// TIA Portal V17 export
// export: Created 2025-03-07T09:19:40.4759984Z, ExportSetting WithDefaults, DisplayName Totally Integrated Automation Portal, DisplayVersion V17 Update 8, DisplayName TIA Portal Openness, DisplayVersion V17 Update 8, DisplayName TIA Portal Version Control Interface, DisplayVersion V17, DisplayName SINAMICS Startdrive Advanced, DisplayVersion V17 SP2, DisplayName SINAMICS Startdrive G110M, G120, G120C, G120D, G120P, G115D, DisplayVersion V17 SP2, DisplayName SINAMICS Startdrive G130, G150, S120, S150, SINAMICS MV, S210, DisplayVersion V17 SP2, DisplayName STEP 7 Professional, DisplayVersion V17 Update 8, DisplayName SINUMERIK ONE STEP 7 Toolbox, DisplayVersion V17 Update 12, DisplayName SINUMERIK 840D sl STEP 7 Toolbox, DisplayVersion V17 Update 12, DisplayName STEP 7 Safety, DisplayVersion V17 Update 6, DisplayName WinCC Advanced, DisplayVersion V17 Update 8
TYPE "M_FUNCTIONS_FIXTURE"
// stored: IsFailsafeCompliant false
   STRUCT
      M_RESET_AUX : Bool;   // RESET AUX
      M_RESET_PULSE : Bool;   // RESET PULSE
      READ_IN_DISABLE_GENERAL : Bool;   // READ-IN DISABLE
      READ_IN_DISABLE_F1 : Bool;   // READ-IN DISABLE
      READ_IN_DISABLE_F2 : Bool;   // READ-IN DISABLE
      SPARE_05 : Bool;
      SPARE_06 : Bool;
      SPARE_07 : Bool;
      M0 : Bool;   // M0-PROGRAMMED STOP (SIEMENS)
      Ack_M0 : Bool;   // ACKNOWLEDGE M0-PROGRAMMED STOP (SIEMENS)
      M1 : Bool;   // M1-OPTIONAL STOP (SIEMENS)
      Ack_M1 : Bool;   // ACKNOWLEDGE M1-OPTIONAL STOP (SIEMENS)
      M2 : Bool;   // M2-END OF PROGRAM, MAIN PROGRAM, AS M30 (SIEMENS)
      Ack_M2 : Bool;   // ACKNOWLEDGE M2-END OF PROGRAM, MAIN PROGRAM, AS M30 (SIEMENS)
      M3 : Bool;   // M3-SPINDLE CLOCKWISE (SIEMENS)
      Ack_M3 : Bool;   // ACKNOWLEDGE M3-SPINDLE CLOCKWISE (SIEMENS)
      M4 : Bool;   // M4-SPINDLE COUNTER CLOCKWISE (SIEMENS)
      Ack_M4 : Bool;   // ACKNOWLEDGE M4-SPINDLE COUNTER CLOCKWISE (SIEMENS)
      M5 : Bool;   // M5-SPINDLE STOP (SIEMENS)
      Ack_M5 : Bool;   // ACKNOWLEDGE M5-SPINDLE STOP (SIEMENS)
      M6 : Bool;   // M6-TOOL CHANGE (SIEMENS)
      Ack_M6 : Bool;   // ACKNOWLEDGE M6-TOOL CHANGE (SIEMENS)
      M7 : Bool;   // M7-
      Ack_M7 : Bool;   // ACKNOWLEDGE M7-
      M8 : Bool;   // M8-
      Ack_M8 : Bool;   // ACKNOWLEDGE M8-
      M9 : Bool;   // M9-
      Ack_M9 : Bool;   // ACKNOWLEDGE M9-
      M10 : Bool;   // M10-
      Ack_M10 : Bool;   // ACKNOWLEDGE M10-
      M11 : Bool;   // M11-
      Ack_M11 : Bool;   // ACKNOWLEDGE M11-
      M12 : Bool;   // M12-
      Ack_M12 : Bool;   // ACKNOWLEDGE M12-
      M13 : Bool;   // M13-
      Ack_M13 : Bool;   // ACKNOWLEDGE M13-
      M14 : Bool;   // M14-
      Ack_M14 : Bool;   // ACKNOWLEDGE M14-
      M15 : Bool;   // M15-
      Ack_M15 : Bool;   // ACKNOWLEDGE M15-
      M16 : Bool;   // M16-
      Ack_M16 : Bool;   // ACKNOWLEDGE M16-
      M17 : Bool;   // M17-END OF SUBPROGRAM (SIEMENS)
      Ack_M17 : Bool;   // ACKNOWLEDGE M17-END OF SUBPROGRAM (SIEMENS)
      M18 : Bool;   // M18-
      Ack_M18 : Bool;   // ACKNOWLEDGE M18-
      M19 : Bool;   // M19-SPINDLE POSITIONING (SIEMENS)
      Ack_M19 : Bool;   // ACKNOWLEDGE M19-SPINDLE POSITIONING (SIEMENS)
      M20 : Bool;   // M20-
      Ack_M20 : Bool;   // ACKNOWLEDGE M20-
      M21 : Bool;   // M21-
      Ack_M21 : Bool;   // ACKNOWLEDGE M21-
      M22 : Bool;   // M22-
      Ack_M22 : Bool;   // ACKNOWLEDGE M22-
      M23 : Bool;   // M23-
      Ack_M23 : Bool;   // ACKNOWLEDGE M23-
      M24 : Bool;   // M24-
      Ack_M24 : Bool;   // ACKNOWLEDGE M24-
      M25 : Bool;   // M25-
      Ack_M25 : Bool;   // ACKNOWLEDGE M25-
      M26 : Bool;   // M26-
      Ack_M26 : Bool;   // ACKNOWLEDGE M26-
      M27 : Bool;   // M27-
      Ack_M27 : Bool;   // ACKNOWLEDGE M27-
      M28 : Bool;   // M28-
      Ack_M28 : Bool;   // ACKNOWLEDGE M28-
      M29 : Bool;   // M29-
      Ack_M29 : Bool;   // ACKNOWLEDGE M29-
      M30 : Bool;   // M30-END OF MAIN PROGRAM (SIEMENS)
      Ack_M30 : Bool;   // ACKNOWLEDGE M30-END OF MAIN PROGRAM (SIEMENS)
      M31 : Bool;   // M31-
      Ack_M31 : Bool;   // ACKNOWLEDGE M31-
      M32 : Bool;   // M32-
      Ack_M32 : Bool;   // ACKNOWLEDGE M32-
      M33 : Bool;   // M33-
      Ack_M33 : Bool;   // ACKNOWLEDGE M33-
      M34 : Bool;   // M34-
      Ack_M34 : Bool;   // ACKNOWLEDGE M34-
      M35 : Bool;   // M35-
      Ack_M35 : Bool;   // ACKNOWLEDGE M35-
      M36 : Bool;   // M36-
      Ack_M36 : Bool;   // ACKNOWLEDGE M36-
      M37 : Bool;   // M37-
      Ack_M37 : Bool;   // ACKNOWLEDGE M37-
      M38 : Bool;   // M38-
      Ack_M38 : Bool;   // ACKNOWLEDGE M38-
      M39 : Bool;   // M39-
      Ack_M39 : Bool;   // ACKNOWLEDGE M39-
      M40 : Bool;   // M40-AUTOMATIC GEAR CHANGE (SIEMENS)
      Ack_M40 : Bool;   // ACKNOWLEDGE M40-AUTOMATIC GEAR CHANGE (SIEMENS)
      M41 : Bool;   // M41-GEAR STAGE 1 (SIEMENS)
      Ack_M41 : Bool;   // ACKNOWLEDGE M41-GEAR STAGE 1 (SIEMENS)
      M42 : Bool;   // M42-GEAR STAGE 2 (SIEMENS)
      Ack_M42 : Bool;   // ACKNOWLEDGE M42-GEAR STAGE 2 (SIEMENS)
      M43 : Bool;   // M43-GEAR STAGE 3 (SIEMENS)
      Ack_M43 : Bool;   // ACKNOWLEDGE M43-GEAR STAGE 3 (SIEMENS)
      M44 : Bool;   // M44-GEAR STAGE 4 (SIEMENS)
      Ack_M44 : Bool;   // ACKNOWLEDGE M44-GEAR STAGE 4 (SIEMENS)
      M45 : Bool;   // M45-GEAR STAGE 5 (SIEMENS)
      Ack_M45 : Bool;   // ACKNOWLEDGE M45-GEAR STAGE 5 (SIEMENS)
      M46 : Bool;   // M46-
      Ack_M46 : Bool;   // ACKNOWLEDGE M46-
      M47 : Bool;   // M47-
      Ack_M47 : Bool;   // ACKNOWLEDGE M47-
      M48 : Bool;   // M48-
      Ack_M48 : Bool;   // ACKNOWLEDGE M48-
      M49 : Bool;   // M49-
      Ack_M49 : Bool;   // ACKNOWLEDGE M49-
      M50 : Bool;   // M50-
      Ack_M50 : Bool;   // ACKNOWLEDGE M50-
      M51 : Bool;   // M51-
      Ack_M51 : Bool;   // ACKNOWLEDGE M51-
      M52 : Bool;   // M52-
      Ack_M52 : Bool;   // ACKNOWLEDGE M52-
      M53 : Bool;   // M53-
      Ack_M53 : Bool;   // ACKNOWLEDGE M53-
      M54 : Bool;   // M54-
      Ack_M54 : Bool;   // ACKNOWLEDGE M54-
      M55 : Bool;   // M55-
      Ack_M55 : Bool;   // ACKNOWLEDGE M55-
      M56 : Bool;   // M56-
      Ack_M56 : Bool;   // ACKNOWLEDGE M56-
      M57 : Bool;   // M57-
      Ack_M57 : Bool;   // ACKNOWLEDGE M57-
      M58 : Bool;   // M58-
      Ack_M58 : Bool;   // ACKNOWLEDGE M58-
      M59 : Bool;   // M59-
      Ack_M59 : Bool;   // ACKNOWLEDGE M59-
      M60 : Bool;   // M60-
      Ack_M60 : Bool;   // ACKNOWLEDGE M60-
      M61 : Bool;   // M61-
      Ack_M61 : Bool;   // ACKNOWLEDGE M61-
      M62 : Bool;   // M62-
      Ack_M62 : Bool;   // ACKNOWLEDGE M62-
      M63 : Bool;   // M63-
      Ack_M63 : Bool;   // ACKNOWLEDGE M63-
      M64 : Bool;   // M64-
      Ack_M64 : Bool;   // ACKNOWLEDGE M64-
      M65 : Bool;   // M65-
      Ack_M65 : Bool;   // ACKNOWLEDGE M65-
      M66 : Bool;   // M66-
      Ack_M66 : Bool;   // ACKNOWLEDGE M66-
      M67 : Bool;   // M67-
      Ack_M67 : Bool;   // ACKNOWLEDGE M67-
      M68 : Bool;   // M68-
      Ack_M68 : Bool;   // ACKNOWLEDGE M68-
      M69 : Bool;   // M69-
      Ack_M69 : Bool;   // ACKNOWLEDGE M69-
      M70 : Bool;   // M70-SPINDLE IS SWITCHED TO AXIS MODE (SIEMENS)
      Ack_M70 : Bool;   // ACKNOWLEDGE M70-SPINDLE IS SWITCHED TO AXIS MODE (SIEMENS)
      M71 : Bool;   // M71-
      Ack_M71 : Bool;   // ACKNOWLEDGE M71-
      M72 : Bool;   // M72-
      Ack_M72 : Bool;   // ACKNOWLEDGE M72-
      M73 : Bool;   // M73-
      Ack_M73 : Bool;   // ACKNOWLEDGE M73-
      M74 : Bool;   // M74-
      Ack_M74 : Bool;   // ACKNOWLEDGE M74-
      M75 : Bool;   // M75-
      Ack_M75 : Bool;   // ACKNOWLEDGE M75-
      M76 : Bool;   // M76-
      Ack_M76 : Bool;   // ACKNOWLEDGE M76-
      M77 : Bool;   // M77-
      Ack_M77 : Bool;   // ACKNOWLEDGE M77-
      M78 : Bool;   // M78-
      Ack_M78 : Bool;   // ACKNOWLEDGE M78-
      M79 : Bool;   // M79-
      Ack_M79 : Bool;   // ACKNOWLEDGE M79-
      M80 : Bool;   // M80-
      Ack_M80 : Bool;   // ACKNOWLEDGE M80-
      M81 : Bool;   // M81-
      Ack_M81 : Bool;   // ACKNOWLEDGE M81-
      M82 : Bool;   // M82-
      Ack_M82 : Bool;   // ACKNOWLEDGE M82-
      M83 : Bool;   // M83-
      Ack_M83 : Bool;   // ACKNOWLEDGE M83-
      M84 : Bool;   // M84-
      Ack_M84 : Bool;   // ACKNOWLEDGE M84-
      M85 : Bool;   // M85-
      Ack_M85 : Bool;   // ACKNOWLEDGE M85-
      M86 : Bool;   // M86-
      Ack_M86 : Bool;   // ACKNOWLEDGE M86-
      M87 : Bool;   // M87-
      Ack_M87 : Bool;   // ACKNOWLEDGE M87-
      M88 : Bool;   // M88-
      Ack_M88 : Bool;   // ACKNOWLEDGE M88-
      M89 : Bool;   // M89-
      Ack_M89 : Bool;   // ACKNOWLEDGE M89-
      M90 : Bool;   // M90-
      Ack_M90 : Bool;   // ACKNOWLEDGE M90-
      M91 : Bool;   // M91-
      Ack_M91 : Bool;   // ACKNOWLEDGE M91-
      M92 : Bool;   // M92-
      Ack_M92 : Bool;   // ACKNOWLEDGE M92-
      M93 : Bool;   // M93-
      Ack_M93 : Bool;   // ACKNOWLEDGE M93-
      M94 : Bool;   // M94-
      Ack_M94 : Bool;   // ACKNOWLEDGE M94-
      M95 : Bool;   // M95-
      Ack_M95 : Bool;   // ACKNOWLEDGE M95-
      M96 : Bool;   // M96-
      Ack_M96 : Bool;   // ACKNOWLEDGE M96-
      M97 : Bool;   // M97-
      Ack_M97 : Bool;   // ACKNOWLEDGE M97-
      M98 : Bool;   // M98-EXTERNAL LANGUAGE (SIEMENS)
      Ack_M98 : Bool;   // ACKNOWLEDGE M98-EXTERNAL LANGUAGE (SIEMENS)
      M99 : Bool;   // M99-EXTERNAL LANGUAGE (SIEMENS)
      Ack_M99 : Bool;   // ACKNOWLEDGE M99-EXTERNAL LANGUAGE (SIEMENS)
      M100 : Bool;   // M100-FIXTURE WAITS FULL DEPTHS UNIT 01R (READ-IN DISABLE)
      Ack_M100 : Bool;   // ACKNOWLEDGE M100-FIXTURE WAITS FULL DEPTHS UNIT 01R (READ-IN DISABLE)
      M101 : Bool;   // M101-FIXTURE WAITS FULL DEPTHS UNIT 01L (READ-IN DISABLE)
      Ack_M101 : Bool;   // ACKNOWLEDGE M101-FIXTURE WAITS FULL DEPTHS UNIT 01L (READ-IN DISABLE)
      M102 : Bool;   // M102-AXIS B IN POSITION DURING LOAD-UNLOAD (READ-IN DISABLE)
      Ack_M102 : Bool;   // ACKNOWLEDGE M102-AXIS B IN POSITION DURING LOAD-UNLOAD (READ-IN DISABLE)
      M103 : Bool;   // M103-
      Ack_M103 : Bool;   // ACKNOWLEDGE M103-
      M104 : Bool;   // M104-
      Ack_M104 : Bool;   // ACKNOWLEDGE M104-
      M105 : Bool;   // M105-
      Ack_M105 : Bool;   // ACKNOWLEDGE M105-
      M106 : Bool;   // M106-
      Ack_M106 : Bool;   // ACKNOWLEDGE M106-
      M107 : Bool;   // M107-
      Ack_M107 : Bool;   // ACKNOWLEDGE M107-
      M108 : Bool;   // M108-
      Ack_M108 : Bool;   // ACKNOWLEDGE M108-
      M109 : Bool;   // M109-
      Ack_M109 : Bool;   // ACKNOWLEDGE M109-
      M110 : Bool;   // M110-UNBLOCK TABLE
      Ack_M110 : Bool;   // ACKNOWLEDGE M110-UNBLOCK TABLE
      M111 : Bool;   // M111-BLOCK TABLE
      Ack_M111 : Bool;   // ACKNOWLEDGE M111-BLOCK TABLE
      M112 : Bool;   // M112-
      Ack_M112 : Bool;   // ACKNOWLEDGE M112-
      M113 : Bool;   // M113-
      Ack_M113 : Bool;   // ACKNOWLEDGE M113-
      M114 : Bool;   // M114-
      Ack_M114 : Bool;   // ACKNOWLEDGE M114-
      M115 : Bool;   // M115-
      Ack_M115 : Bool;   // ACKNOWLEDGE M115-
      M116 : Bool;   // M116-
      Ack_M116 : Bool;   // ACKNOWLEDGE M116-
      M117 : Bool;   // M117-
      Ack_M117 : Bool;   // ACKNOWLEDGE M117-
      M118 : Bool;   // M118-
      Ack_M118 : Bool;   // ACKNOWLEDGE M118-
      M119 : Bool;   // M119-
      Ack_M119 : Bool;   // ACKNOWLEDGE M119-
      M120 : Bool;   // M120-
      Ack_M120 : Bool;   // ACKNOWLEDGE M120-
      M121 : Bool;   // M121-
      Ack_M121 : Bool;   // ACKNOWLEDGE M121-
      M122 : Bool;   // M122-
      Ack_M122 : Bool;   // ACKNOWLEDGE M122-
      M123 : Bool;   // M123-AXIS B TORQUE LIMIT EXCEEDED
      Ack_M123 : Bool;   // ACKNOWLEDGE M123-AXIS B TORQUE LIMIT EXCEEDED
      M124 : Bool;   // M124-
      Ack_M124 : Bool;   // ACKNOWLEDGE M124-
      M125 : Bool;   // M125-
      Ack_M125 : Bool;   // ACKNOWLEDGE M125-
      M126 : Bool;   // M126-
      Ack_M126 : Bool;   // ACKNOWLEDGE M126-
      M127 : Bool;   // M127-
      Ack_M127 : Bool;   // ACKNOWLEDGE M127-
      M128 : Bool;   // M128-
      Ack_M128 : Bool;   // ACKNOWLEDGE M128-
      M129 : Bool;   // M129-
      Ack_M129 : Bool;   // ACKNOWLEDGE M129-
      M130 : Bool;   // M130-
      Ack_M130 : Bool;   // ACKNOWLEDGE M130-
      M131 : Bool;   // M131-
      Ack_M131 : Bool;   // ACKNOWLEDGE M131-
      M132 : Bool;   // M132-
      Ack_M132 : Bool;   // ACKNOWLEDGE M132-
      M133 : Bool;   // M133-
      Ack_M133 : Bool;   // ACKNOWLEDGE M133-
      M134 : Bool;   // M134-
      Ack_M134 : Bool;   // ACKNOWLEDGE M134-
      M135 : Bool;   // M135-
      Ack_M135 : Bool;   // ACKNOWLEDGE M135-
      M136 : Bool;   // M136-
      Ack_M136 : Bool;   // ACKNOWLEDGE M136-
      M137 : Bool;   // M137-
      Ack_M137 : Bool;   // ACKNOWLEDGE M137-
      M138 : Bool;   // M138-
      Ack_M138 : Bool;   // ACKNOWLEDGE M138-
      M139 : Bool;   // M139-
      Ack_M139 : Bool;   // ACKNOWLEDGE M139-
      M140 : Bool;   // M140-
      Ack_M140 : Bool;   // ACKNOWLEDGE M140-
      M141 : Bool;   // M141-
      Ack_M141 : Bool;   // ACKNOWLEDGE M141-
      M142 : Bool;   // M142-
      Ack_M142 : Bool;   // ACKNOWLEDGE M142-
      M143 : Bool;   // M143-
      Ack_M143 : Bool;   // ACKNOWLEDGE M143-
      M144 : Bool;   // M144-
      Ack_M144 : Bool;   // ACKNOWLEDGE M144-
      M145 : Bool;   // M145-
      Ack_M145 : Bool;   // ACKNOWLEDGE M145-
      M146 : Bool;   // M146-
      Ack_M146 : Bool;   // ACKNOWLEDGE M146-
      M147 : Bool;   // M147-
      Ack_M147 : Bool;   // ACKNOWLEDGE M147-
      M148 : Bool;   // M148-
      Ack_M148 : Bool;   // ACKNOWLEDGE M148-
      M149 : Bool;   // M149-
      Ack_M149 : Bool;   // ACKNOWLEDGE M149-
      M150 : Bool;   // M150-AUTOMATIC DOOR OPEN
      Ack_M150 : Bool;   // ACKNOWLEDGE M150-AUTOMATIC DOOR OPEN
      M151 : Bool;   // M151-AUTOMATIC DOOR CLOSE
      Ack_M151 : Bool;   // ACKNOWLEDGE M151-AUTOMATIC DOOR CLOSE
      M152 : Bool;   // M152-
      Ack_M152 : Bool;   // ACKNOWLEDGE M152-
      M153 : Bool;   // M153-
      Ack_M153 : Bool;   // ACKNOWLEDGE M153-
      M154 : Bool;   // M154-
      Ack_M154 : Bool;   // ACKNOWLEDGE M154-
      M155 : Bool;   // M155-
      Ack_M155 : Bool;   // ACKNOWLEDGE M155-
      M156 : Bool;   // M156-
      Ack_M156 : Bool;   // ACKNOWLEDGE M156-
      M157 : Bool;   // M157-
      Ack_M157 : Bool;   // ACKNOWLEDGE M157-
      M158 : Bool;   // M158-
      Ack_M158 : Bool;   // ACKNOWLEDGE M158-
      M159 : Bool;   // M159-
      Ack_M159 : Bool;   // ACKNOWLEDGE M159-
      M160 : Bool;   // M160-
      Ack_M160 : Bool;   // ACKNOWLEDGE M160-
      M161 : Bool;   // M161-
      Ack_M161 : Bool;   // ACKNOWLEDGE M161-
      M162 : Bool;   // M162-
      Ack_M162 : Bool;   // ACKNOWLEDGE M162-
      M163 : Bool;   // M163-
      Ack_M163 : Bool;   // ACKNOWLEDGE M163-
      M164 : Bool;   // M164-
      Ack_M164 : Bool;   // ACKNOWLEDGE M164-
      M165 : Bool;   // M165-
      Ack_M165 : Bool;   // ACKNOWLEDGE M165-
      M166 : Bool;   // M166-
      Ack_M166 : Bool;   // ACKNOWLEDGE M166-
      M167 : Bool;   // M167-
      Ack_M167 : Bool;   // ACKNOWLEDGE M167-
      M168 : Bool;   // M168-
      Ack_M168 : Bool;   // ACKNOWLEDGE M168-
      M169 : Bool;   // M169-
      Ack_M169 : Bool;   // ACKNOWLEDGE M169-
      M170 : Bool;   // M170-
      Ack_M170 : Bool;   // ACKNOWLEDGE M170-
      M171 : Bool;   // M171-
      Ack_M171 : Bool;   // ACKNOWLEDGE M171-
      M172 : Bool;   // M172-
      Ack_M172 : Bool;   // ACKNOWLEDGE M172-
      M173 : Bool;   // M173-
      Ack_M173 : Bool;   // ACKNOWLEDGE M173-
      M174 : Bool;   // M174-
      Ack_M174 : Bool;   // ACKNOWLEDGE M174-
      M175 : Bool;   // M175-
      Ack_M175 : Bool;   // ACKNOWLEDGE M175-
      M176 : Bool;   // M176-
      Ack_M176 : Bool;   // ACKNOWLEDGE M176-
      M177 : Bool;   // M177-
      Ack_M177 : Bool;   // ACKNOWLEDGE M177-
      M178 : Bool;   // M178-
      Ack_M178 : Bool;   // ACKNOWLEDGE M178-
      M179 : Bool;   // M179-
      Ack_M179 : Bool;   // ACKNOWLEDGE M179-
      M180 : Bool;   // M180-
      Ack_M180 : Bool;   // ACKNOWLEDGE M180-
      M181 : Bool;   // M181-
      Ack_M181 : Bool;   // ACKNOWLEDGE M181-
      M182 : Bool;   // M182-
      Ack_M182 : Bool;   // ACKNOWLEDGE M182-
      M183 : Bool;   // M183-
      Ack_M183 : Bool;   // ACKNOWLEDGE M183-
      M184 : Bool;   // M184-
      Ack_M184 : Bool;   // ACKNOWLEDGE M184-
      M185 : Bool;   // M185-
      Ack_M185 : Bool;   // ACKNOWLEDGE M185-
      M186 : Bool;   // M186-
      Ack_M186 : Bool;   // ACKNOWLEDGE M186-
      M187 : Bool;   // M187-
      Ack_M187 : Bool;   // ACKNOWLEDGE M187-
      M188 : Bool;   // M188-
      Ack_M188 : Bool;   // ACKNOWLEDGE M188-
      M189 : Bool;   // M189-
      Ack_M189 : Bool;   // ACKNOWLEDGE M189-
      M190 : Bool;   // M190-
      Ack_M190 : Bool;   // ACKNOWLEDGE M190-
      M191 : Bool;   // M191-
      Ack_M191 : Bool;   // ACKNOWLEDGE M191-
      M192 : Bool;   // M192-
      Ack_M192 : Bool;   // ACKNOWLEDGE M192-
      M193 : Bool;   // M193-
      Ack_M193 : Bool;   // ACKNOWLEDGE M193-
      M194 : Bool;   // M194-
      Ack_M194 : Bool;   // ACKNOWLEDGE M194-
      M195 : Bool;   // M195-
      Ack_M195 : Bool;   // ACKNOWLEDGE M195-
      M196 : Bool;   // M196-
      Ack_M196 : Bool;   // ACKNOWLEDGE M196-
      M197 : Bool;   // M197-
      Ack_M197 : Bool;   // ACKNOWLEDGE M197-
      M198 : Bool;   // M198-
      Ack_M198 : Bool;   // ACKNOWLEDGE M198-
      M199 : Bool;   // M199-
      Ack_M199 : Bool;   // ACKNOWLEDGE M199-
      M200 : Bool;   // M200-
      Ack_M200 : Bool;   // ACKNOWLEDGE M200-
      M201 : Bool;   // M201-
      Ack_M201 : Bool;   // ACKNOWLEDGE M201-
      M202 : Bool;   // M202-
      Ack_M202 : Bool;   // ACKNOWLEDGE M202-
      M203 : Bool;   // M203-
      Ack_M203 : Bool;   // ACKNOWLEDGE M203-
      M204 : Bool;   // M204-
      Ack_M204 : Bool;   // ACKNOWLEDGE M204-
      M205 : Bool;   // M205-
      Ack_M205 : Bool;   // ACKNOWLEDGE M205-
      M206 : Bool;   // M206-
      Ack_M206 : Bool;   // ACKNOWLEDGE M206-
      M207 : Bool;   // M207-
      Ack_M207 : Bool;   // ACKNOWLEDGE M207-
      M208 : Bool;   // M208-
      Ack_M208 : Bool;   // ACKNOWLEDGE M208-
      M209 : Bool;   // M209-
      Ack_M209 : Bool;   // ACKNOWLEDGE M209-
      M210 : Bool;   // M210-
      Ack_M210 : Bool;   // ACKNOWLEDGE M210-
      M211 : Bool;   // M211-
      Ack_M211 : Bool;   // ACKNOWLEDGE M211-
      M212 : Bool;   // M212-
      Ack_M212 : Bool;   // ACKNOWLEDGE M212-
      M213 : Bool;   // M213-
      Ack_M213 : Bool;   // ACKNOWLEDGE M213-
      M214 : Bool;   // M214-
      Ack_M214 : Bool;   // ACKNOWLEDGE M214-
      M215 : Bool;   // M215-
      Ack_M215 : Bool;   // ACKNOWLEDGE M215-
      M216 : Bool;   // M216-
      Ack_M216 : Bool;   // ACKNOWLEDGE M216-
      M217 : Bool;   // M217-
      Ack_M217 : Bool;   // ACKNOWLEDGE M217-
      M218 : Bool;   // M218-
      Ack_M218 : Bool;   // ACKNOWLEDGE M218-
      M219 : Bool;   // M219-
      Ack_M219 : Bool;   // ACKNOWLEDGE M219-
      M220 : Bool;   // M220-
      Ack_M220 : Bool;   // ACKNOWLEDGE M220-
      M221 : Bool;   // M221-
      Ack_M221 : Bool;   // ACKNOWLEDGE M221-
      M222 : Bool;   // M222-
      Ack_M222 : Bool;   // ACKNOWLEDGE M222-
      M223 : Bool;   // M223-
      Ack_M223 : Bool;   // ACKNOWLEDGE M223-
      M224 : Bool;   // M224-
      Ack_M224 : Bool;   // ACKNOWLEDGE M224-
      M225 : Bool;   // M225-
      Ack_M225 : Bool;   // ACKNOWLEDGE M225-
      M226 : Bool;   // M226-
      Ack_M226 : Bool;   // ACKNOWLEDGE M226-
      M227 : Bool;   // M227-
      Ack_M227 : Bool;   // ACKNOWLEDGE M227-
      M228 : Bool;   // M228-
      Ack_M228 : Bool;   // ACKNOWLEDGE M228-
      M229 : Bool;   // M229-
      Ack_M229 : Bool;   // ACKNOWLEDGE M229-
      M230 : Bool;   // M230-
      Ack_M230 : Bool;   // ACKNOWLEDGE M230-
      M231 : Bool;   // M231-
      Ack_M231 : Bool;   // ACKNOWLEDGE M231-
      M232 : Bool;   // M232-
      Ack_M232 : Bool;   // ACKNOWLEDGE M232-
      M233 : Bool;   // M233-
      Ack_M233 : Bool;   // ACKNOWLEDGE M233-
      M234 : Bool;   // M234-
      Ack_M234 : Bool;   // ACKNOWLEDGE M234-
      M235 : Bool;   // M235-
      Ack_M235 : Bool;   // ACKNOWLEDGE M235-
      M236 : Bool;   // M236-
      Ack_M236 : Bool;   // ACKNOWLEDGE M236-
      M237 : Bool;   // M237-
      Ack_M237 : Bool;   // ACKNOWLEDGE M237-
      M238 : Bool;   // M238-
      Ack_M238 : Bool;   // ACKNOWLEDGE M238-
      M239 : Bool;   // M239-
      Ack_M239 : Bool;   // ACKNOWLEDGE M239-
      M240 : Bool;   // M240-
      Ack_M240 : Bool;   // ACKNOWLEDGE M240-
      M241 : Bool;   // M241-
      Ack_M241 : Bool;   // ACKNOWLEDGE M241-
      M242 : Bool;   // M242-
      Ack_M242 : Bool;   // ACKNOWLEDGE M242-
      M243 : Bool;   // M243-
      Ack_M243 : Bool;   // ACKNOWLEDGE M243-
      M244 : Bool;   // M244-
      Ack_M244 : Bool;   // ACKNOWLEDGE M244-
      M245 : Bool;   // M245-
      Ack_M245 : Bool;   // ACKNOWLEDGE M245-
      M246 : Bool;   // M246-
      Ack_M246 : Bool;   // ACKNOWLEDGE M246-
      M247 : Bool;   // M247-
      Ack_M247 : Bool;   // ACKNOWLEDGE M247-
      M248 : Bool;   // M248-
      Ack_M248 : Bool;   // ACKNOWLEDGE M248-
      M249 : Bool;   // M249-
      Ack_M249 : Bool;   // ACKNOWLEDGE M249-
      M250 : Bool;   // M250-
      Ack_M250 : Bool;   // ACKNOWLEDGE M250-
      M251 : Bool;   // M251-
      Ack_M251 : Bool;   // ACKNOWLEDGE M251-
      M252 : Bool;   // M252-
      Ack_M252 : Bool;   // ACKNOWLEDGE M252-
      M253 : Bool;   // M253-
      Ack_M253 : Bool;   // ACKNOWLEDGE M253-
      M254 : Bool;   // M254-
      Ack_M254 : Bool;   // ACKNOWLEDGE M254-
      M255 : Bool;   // M255-
      Ack_M255 : Bool;   // ACKNOWLEDGE M255-
      M256 : Bool;   // M256-
      Ack_M256 : Bool;   // ACKNOWLEDGE M256-
      M257 : Bool;   // M257-
      Ack_M257 : Bool;   // ACKNOWLEDGE M257-
      M258 : Bool;   // M258-
      Ack_M258 : Bool;   // ACKNOWLEDGE M258-
      M259 : Bool;   // M259-
      Ack_M259 : Bool;   // ACKNOWLEDGE M259-
      M260 : Bool;   // M260-
      Ack_M260 : Bool;   // ACKNOWLEDGE M260-
      M261 : Bool;   // M261-
      Ack_M261 : Bool;   // ACKNOWLEDGE M261-
      M262 : Bool;   // M262-
      Ack_M262 : Bool;   // ACKNOWLEDGE M262-
      M263 : Bool;   // M263-
      Ack_M263 : Bool;   // ACKNOWLEDGE M263-
      M264 : Bool;   // M264-
      Ack_M264 : Bool;   // ACKNOWLEDGE M264-
      M265 : Bool;   // M265-
      Ack_M265 : Bool;   // ACKNOWLEDGE M265-
      M266 : Bool;   // M266-
      Ack_M266 : Bool;   // ACKNOWLEDGE M266-
      M267 : Bool;   // M267-
      Ack_M267 : Bool;   // ACKNOWLEDGE M267-
      M268 : Bool;   // M268-
      Ack_M268 : Bool;   // ACKNOWLEDGE M268-
      M269 : Bool;   // M269-
      Ack_M269 : Bool;   // ACKNOWLEDGE M269-
      M270 : Bool;   // M270-
      Ack_M270 : Bool;   // ACKNOWLEDGE M270-
      M271 : Bool;   // M271-
      Ack_M271 : Bool;   // ACKNOWLEDGE M271-
      M272 : Bool;   // M272-
      Ack_M272 : Bool;   // ACKNOWLEDGE M272-
      M273 : Bool;   // M273-
      Ack_M273 : Bool;   // ACKNOWLEDGE M273-
      M274 : Bool;   // M274-
      Ack_M274 : Bool;   // ACKNOWLEDGE M274-
      M275 : Bool;   // M275-
      Ack_M275 : Bool;   // ACKNOWLEDGE M275-
      M276 : Bool;   // M276-
      Ack_M276 : Bool;   // ACKNOWLEDGE M276-
      M277 : Bool;   // M277-
      Ack_M277 : Bool;   // ACKNOWLEDGE M277-
      M278 : Bool;   // M278-
      Ack_M278 : Bool;   // ACKNOWLEDGE M278-
      M279 : Bool;   // M279-
      Ack_M279 : Bool;   // ACKNOWLEDGE M279-
      M280 : Bool;   // M280-
      Ack_M280 : Bool;   // ACKNOWLEDGE M280-
      M281 : Bool;   // M281-
      Ack_M281 : Bool;   // ACKNOWLEDGE M281-
      M282 : Bool;   // M282-
      Ack_M282 : Bool;   // ACKNOWLEDGE M282-
      M283 : Bool;   // M283-
      Ack_M283 : Bool;   // ACKNOWLEDGE M283-
      M284 : Bool;   // M284-
      Ack_M284 : Bool;   // ACKNOWLEDGE M284-
      M285 : Bool;   // M285-
      Ack_M285 : Bool;   // ACKNOWLEDGE M285-
      M286 : Bool;   // M286-
      Ack_M286 : Bool;   // ACKNOWLEDGE M286-
      M287 : Bool;   // M287-
      Ack_M287 : Bool;   // ACKNOWLEDGE M287-
      M288 : Bool;   // M288-
      Ack_M288 : Bool;   // ACKNOWLEDGE M288-
      M289 : Bool;   // M289-
      Ack_M289 : Bool;   // ACKNOWLEDGE M289-
      M290 : Bool;   // M290-
      Ack_M290 : Bool;   // ACKNOWLEDGE M290-
      M291 : Bool;   // M291-
      Ack_M291 : Bool;   // ACKNOWLEDGE M291-
      M292 : Bool;   // M292-
      Ack_M292 : Bool;   // ACKNOWLEDGE M292-
      M293 : Bool;   // M293-
      Ack_M293 : Bool;   // ACKNOWLEDGE M293-
      M294 : Bool;   // M294-
      Ack_M294 : Bool;   // ACKNOWLEDGE M294-
      M295 : Bool;   // M295-
      Ack_M295 : Bool;   // ACKNOWLEDGE M295-
      M296 : Bool;   // M296-
      Ack_M296 : Bool;   // ACKNOWLEDGE M296-
      M297 : Bool;   // M297-
      Ack_M297 : Bool;   // ACKNOWLEDGE M297-
      M298 : Bool;   // M298-
      Ack_M298 : Bool;   // ACKNOWLEDGE M298-
      M299 : Bool;   // M299-
      Ack_M299 : Bool;   // ACKNOWLEDGE M299-
      M300 : Bool;   // M300-
      Ack_M300 : Bool;   // ACKNOWLEDGE M300-
      M301 : Bool;   // M301-
      Ack_M301 : Bool;   // ACKNOWLEDGE M301-
      M302 : Bool;   // M302-
      Ack_M302 : Bool;   // ACKNOWLEDGE M302-
      M303 : Bool;   // M303-
      Ack_M303 : Bool;   // ACKNOWLEDGE M303-
      M304 : Bool;   // M304-
      Ack_M304 : Bool;   // ACKNOWLEDGE M304-
      M305 : Bool;   // M305-
      Ack_M305 : Bool;   // ACKNOWLEDGE M305-
      M306 : Bool;   // M306-
      Ack_M306 : Bool;   // ACKNOWLEDGE M306-
      M307 : Bool;   // M307-
      Ack_M307 : Bool;   // ACKNOWLEDGE M307-
      M308 : Bool;   // M308-
      Ack_M308 : Bool;   // ACKNOWLEDGE M308-
      M309 : Bool;   // M309-
      Ack_M309 : Bool;   // ACKNOWLEDGE M309-
      M310 : Bool;   // M310-
      Ack_M310 : Bool;   // ACKNOWLEDGE M310-
      M311 : Bool;   // M311-
      Ack_M311 : Bool;   // ACKNOWLEDGE M311-
      M312 : Bool;   // M312-
      Ack_M312 : Bool;   // ACKNOWLEDGE M312-
      M313 : Bool;   // M313-
      Ack_M313 : Bool;   // ACKNOWLEDGE M313-
      M314 : Bool;   // M314-
      Ack_M314 : Bool;   // ACKNOWLEDGE M314-
      M315 : Bool;   // M315-
      Ack_M315 : Bool;   // ACKNOWLEDGE M315-
      M316 : Bool;   // M316-
      Ack_M316 : Bool;   // ACKNOWLEDGE M316-
      M317 : Bool;   // M317-
      Ack_M317 : Bool;   // ACKNOWLEDGE M317-
      M318 : Bool;   // M318-
      Ack_M318 : Bool;   // ACKNOWLEDGE M318-
      M319 : Bool;   // M319-
      Ack_M319 : Bool;   // ACKNOWLEDGE M319-
      M320 : Bool;   // M320-MACHINE FLUSH VALVE SWITCH ON
      Ack_M320 : Bool;   // ACKNOWLEDGE M320-MACHINE FLUSH VALVE SWITCH ON
      M321 : Bool;   // M321-MACHINE FLUSH VALVE SWITCH OFF
      Ack_M321 : Bool;   // ACKNOWLEDGE M321-MACHINE FLUSH VALVE SWITCH OFF
      M322 : Bool;   // M322-
      Ack_M322 : Bool;   // ACKNOWLEDGE M322-
      M323 : Bool;   // M323-
      Ack_M323 : Bool;   // ACKNOWLEDGE M323-
      M324 : Bool;   // M324-FIXTURE 1 CLEANING VALVE SWITCH ON
      Ack_M324 : Bool;   // ACKNOWLEDGE M324-FIXTURE 1 CLEANING VALVE SWITCH ON
      M325 : Bool;   // M325-FIXTURE 1 CLEANING VALVE SWITCH OFF
      Ack_M325 : Bool;   // ACKNOWLEDGE M325-FIXTURE 1 CLEANING VALVE SWITCH OFF
      M326 : Bool;   // M326-FIXTURE 2 CLEANING VALVE SWITCH ON
      Ack_M326 : Bool;   // ACKNOWLEDGE M326-FIXTURE 2 CLEANING VALVE SWITCH ON
      M327 : Bool;   // M327-FIXTURE 2 CLEANING VALVE SWITCH OFF
      Ack_M327 : Bool;   // ACKNOWLEDGE M327-FIXTURE 2 CLEANING VALVE SWITCH OFF
      M328 : Bool;   // M328-
      Ack_M328 : Bool;   // ACKNOWLEDGE M328-
      M329 : Bool;   // M329-
      Ack_M329 : Bool;   // ACKNOWLEDGE M329-
      M330 : Bool;   // M330-
      Ack_M330 : Bool;   // ACKNOWLEDGE M330-
      M331 : Bool;   // M331-
      Ack_M331 : Bool;   // ACKNOWLEDGE M331-
      M332 : Bool;   // M332-FIXTURE 1 INTERNAL BLOWING SWITCH ON
      Ack_M332 : Bool;   // ACKNOWLEDGE M332-FIXTURE 1 INTERNAL BLOWING SWITCH ON
      M333 : Bool;   // M333-FIXTURE 1 INTERNAL BLOWING SWITCH OFF
      Ack_M333 : Bool;   // ACKNOWLEDGE M333-FIXTURE 1 INTERNAL BLOWING SWITCH OFF
      M334 : Bool;   // M334-FIXTURE 2 INTERNAL BLOWING SWITCH ON
      Ack_M334 : Bool;   // ACKNOWLEDGE M334-FIXTURE 2 INTERNAL BLOWING SWITCH ON
      M335 : Bool;   // M335-FIXTURE 2 INTERNAL BLOWING SWITCH OFF
      Ack_M335 : Bool;   // ACKNOWLEDGE M335-FIXTURE 2 INTERNAL BLOWING SWITCH OFF
      M336 : Bool;   // M336-
      Ack_M336 : Bool;   // ACKNOWLEDGE M336-
      M337 : Bool;   // M337-
      Ack_M337 : Bool;   // ACKNOWLEDGE M337-
      M338 : Bool;   // M338-
      Ack_M338 : Bool;   // ACKNOWLEDGE M338-
      M339 : Bool;   // M339-
      Ack_M339 : Bool;   // ACKNOWLEDGE M339-
      M340 : Bool;   // M340-
      Ack_M340 : Bool;   // ACKNOWLEDGE M340-
      M341 : Bool;   // M341-
      Ack_M341 : Bool;   // ACKNOWLEDGE M341-
      M342 : Bool;   // M342-
      Ack_M342 : Bool;   // ACKNOWLEDGE M342-
      M343 : Bool;   // M343-
      Ack_M343 : Bool;   // ACKNOWLEDGE M343-
      M344 : Bool;   // M344-
      Ack_M344 : Bool;   // ACKNOWLEDGE M344-
      M345 : Bool;   // M345-
      Ack_M345 : Bool;   // ACKNOWLEDGE M345-
      M346 : Bool;   // M346-
      Ack_M346 : Bool;   // ACKNOWLEDGE M346-
      M347 : Bool;   // M347-
      Ack_M347 : Bool;   // ACKNOWLEDGE M347-
      M348 : Bool;   // M348-
      Ack_M348 : Bool;   // ACKNOWLEDGE M348-
      M349 : Bool;   // M349-
      Ack_M349 : Bool;   // ACKNOWLEDGE M349-
      M350 : Bool;   // M350-
      Ack_M350 : Bool;   // ACKNOWLEDGE M350-
      M351 : Bool;   // M351-
      Ack_M351 : Bool;   // ACKNOWLEDGE M351-
      M352 : Bool;   // M352-
      Ack_M352 : Bool;   // ACKNOWLEDGE M352-
      M353 : Bool;   // M353-
      Ack_M353 : Bool;   // ACKNOWLEDGE M353-
      M354 : Bool;   // M354-
      Ack_M354 : Bool;   // ACKNOWLEDGE M354-
      M355 : Bool;   // M355-
      Ack_M355 : Bool;   // ACKNOWLEDGE M355-
      M356 : Bool;   // M356-
      Ack_M356 : Bool;   // ACKNOWLEDGE M356-
      M357 : Bool;   // M357-
      Ack_M357 : Bool;   // ACKNOWLEDGE M357-
      M358 : Bool;   // M358-
      Ack_M358 : Bool;   // ACKNOWLEDGE M358-
      M359 : Bool;   // M359-
      Ack_M359 : Bool;   // ACKNOWLEDGE M359-
      M360 : Bool;   // M360-
      Ack_M360 : Bool;   // ACKNOWLEDGE M360-
      M361 : Bool;   // M361-
      Ack_M361 : Bool;   // ACKNOWLEDGE M361-
      M362 : Bool;   // M362-
      Ack_M362 : Bool;   // ACKNOWLEDGE M362-
      M363 : Bool;   // M363-
      Ack_M363 : Bool;   // ACKNOWLEDGE M363-
      M364 : Bool;   // M364-
      Ack_M364 : Bool;   // ACKNOWLEDGE M364-
      M365 : Bool;   // M365-
      Ack_M365 : Bool;   // ACKNOWLEDGE M365-
      M366 : Bool;   // M366-
      Ack_M366 : Bool;   // ACKNOWLEDGE M366-
      M367 : Bool;   // M367-
      Ack_M367 : Bool;   // ACKNOWLEDGE M367-
      M368 : Bool;   // M368-
      Ack_M368 : Bool;   // ACKNOWLEDGE M368-
      M369 : Bool;   // M369-
      Ack_M369 : Bool;   // ACKNOWLEDGE M369-
      M370 : Bool;   // M370-
      Ack_M370 : Bool;   // ACKNOWLEDGE M370-
      M371 : Bool;   // M371-
      Ack_M371 : Bool;   // ACKNOWLEDGE M371-
      M372 : Bool;   // M372-
      Ack_M372 : Bool;   // ACKNOWLEDGE M372-
      M373 : Bool;   // M373-
      Ack_M373 : Bool;   // ACKNOWLEDGE M373-
      M374 : Bool;   // M374-
      Ack_M374 : Bool;   // ACKNOWLEDGE M374-
      M375 : Bool;   // M375-
      Ack_M375 : Bool;   // ACKNOWLEDGE M375-
      M376 : Bool;   // M376-
      Ack_M376 : Bool;   // ACKNOWLEDGE M376-
      M377 : Bool;   // M377-
      Ack_M377 : Bool;   // ACKNOWLEDGE M377-
      M378 : Bool;   // M378-
      Ack_M378 : Bool;   // ACKNOWLEDGE M378-
      M379 : Bool;   // M379-
      Ack_M379 : Bool;   // ACKNOWLEDGE M379-
      M380 : Bool;   // M380-
      Ack_M380 : Bool;   // ACKNOWLEDGE M380-
      M381 : Bool;   // M381-
      Ack_M381 : Bool;   // ACKNOWLEDGE M381-
      M382 : Bool;   // M382-
      Ack_M382 : Bool;   // ACKNOWLEDGE M382-
      M383 : Bool;   // M383-
      Ack_M383 : Bool;   // ACKNOWLEDGE M383-
      M384 : Bool;   // M384-
      Ack_M384 : Bool;   // ACKNOWLEDGE M384-
      M385 : Bool;   // M385-
      Ack_M385 : Bool;   // ACKNOWLEDGE M385-
      M386 : Bool;   // M386-
      Ack_M386 : Bool;   // ACKNOWLEDGE M386-
      M387 : Bool;   // M387-
      Ack_M387 : Bool;   // ACKNOWLEDGE M387-
      M388 : Bool;   // M388-
      Ack_M388 : Bool;   // ACKNOWLEDGE M388-
      M389 : Bool;   // M389-
      Ack_M389 : Bool;   // ACKNOWLEDGE M389-
      M390 : Bool;   // M390-
      Ack_M390 : Bool;   // ACKNOWLEDGE M390-
      M391 : Bool;   // M391-
      Ack_M391 : Bool;   // ACKNOWLEDGE M391-
      M392 : Bool;   // M392-
      Ack_M392 : Bool;   // ACKNOWLEDGE M392-
      M393 : Bool;   // M393-
      Ack_M393 : Bool;   // ACKNOWLEDGE M393-
      M394 : Bool;   // M394-
      Ack_M394 : Bool;   // ACKNOWLEDGE M394-
      M395 : Bool;   // M395-
      Ack_M395 : Bool;   // ACKNOWLEDGE M395-
      M396 : Bool;   // M396-
      Ack_M396 : Bool;   // ACKNOWLEDGE M396-
      M397 : Bool;   // M397-
      Ack_M397 : Bool;   // ACKNOWLEDGE M397-
      M398 : Bool;   // M398-
      Ack_M398 : Bool;   // ACKNOWLEDGE M398-
      M399 : Bool;   // M399-
      Ack_M399 : Bool;   // ACKNOWLEDGE M399-
      M400 : Bool;   // M400-FIXTURE 1 CLAMP SEQUENCE (READ-IN DISABLE)
      Ack_M400 : Bool;   // ACKNOWLEDGE M400-FIXTURE 1 CLAMP SEQUENCE (READ-IN DISABLE)
      M401 : Bool;   // M401-FIXTURE 1 CLAMP SEQUENCE
      Ack_M401 : Bool;   // ACKNOWLEDGE M401-FIXTURE 1 CLAMP SEQUENCE
      M402 : Bool;   // M402-FIXTURE 1 UNCLAMP SEQUENCE (READ-IN DISABLE)
      Ack_M402 : Bool;   // ACKNOWLEDGE M402-FIXTURE 1 UNCLAMP SEQUENCE (READ-IN DISABLE)
      M403 : Bool;   // M403-FIXTURE 1 UNCLAMP SEQUENCE
      Ack_M403 : Bool;   // ACKNOWLEDGE M403-FIXTURE 1 UNCLAMP SEQUENCE
      M404 : Bool;   // M404-FIXTURE 1 VERIFY PART AND TOOL IS CLAMPED DURING MACHINING (WHEN TRUE DO). TOGGLED
      Ack_M404 : Bool;   // ACKNOWLEDGE M404-FIXTURE 1 VERIFY PART AND TOOL IS CLAMPED DURING MACHINING (WHEN TRUE DO). TOGGLED
      M405 : Bool;   // M405-FIXTURE 1 VERIFY PART AND TOOL IS CLAMPED LOW PRESSURE DURING MACHINING (WHEN TRUE DO). TOGGLED
      Ack_M405 : Bool;   // ACKNOWLEDGE M405-FIXTURE 1 VERIFY PART AND TOOL IS CLAMPED LOW PRESSURE DURING MACHINING (WHEN TRUE DO). TOGGLED
      M406 : Bool;   // M406-FIXTURE 1 VERIFY PARTS ARE UNCLAMPED PARTS LOADING (WHEN TRUE DO). TOGGLED
      Ack_M406 : Bool;   // ACKNOWLEDGE M406-FIXTURE 1 VERIFY PARTS ARE UNCLAMPED PARTS LOADING (WHEN TRUE DO). TOGGLED
      M407 : Bool;   // M407-FIXTURE 1 VERIFY FIXTURE REMAINS CLAMPED
      Ack_M407 : Bool;   // ACKNOWLEDGE M407-FIXTURE 1 VERIFY FIXTURE REMAINS CLAMPED
      M408 : Bool;   // M408-
      Ack_M408 : Bool;   // ACKNOWLEDGE M408-
      M409 : Bool;   // M409-
      Ack_M409 : Bool;   // ACKNOWLEDGE M409-
      M410 : Bool;   // M410-
      Ack_M410 : Bool;   // ACKNOWLEDGE M410-
      M411 : Bool;   // M411-
      Ack_M411 : Bool;   // ACKNOWLEDGE M411-
      M412 : Bool;   // M412-
      Ack_M412 : Bool;   // ACKNOWLEDGE M412-
      M413 : Bool;   // M413-
      Ack_M413 : Bool;   // ACKNOWLEDGE M413-
      M414 : Bool;   // M414-
      Ack_M414 : Bool;   // ACKNOWLEDGE M414-
      M415 : Bool;   // M415-
      Ack_M415 : Bool;   // ACKNOWLEDGE M415-
      M416 : Bool;   // M416-
      Ack_M416 : Bool;   // ACKNOWLEDGE M416-
      M417 : Bool;   // M417-
      Ack_M417 : Bool;   // ACKNOWLEDGE M417-
      M418 : Bool;   // M418-
      Ack_M418 : Bool;   // ACKNOWLEDGE M418-
      M419 : Bool;   // M419-
      Ack_M419 : Bool;   // ACKNOWLEDGE M419-
      M420 : Bool;   // M420-FIXTURE 1 AXIAL LOCATOR LOCATE (READ-IN DISABLE)
      Ack_M420 : Bool;   // ACKNOWLEDGE M420-FIXTURE 1 AXIAL LOCATOR LOCATE (READ-IN DISABLE)
      M421 : Bool;   // M421-FIXTURE 1 AXIAL LOCATOR LOCATE
      Ack_M421 : Bool;   // ACKNOWLEDGE M421-FIXTURE 1 AXIAL LOCATOR LOCATE
      M422 : Bool;   // M422-FIXTURE 1 AXIAL LOCATOR RETURN (READ-IN DISABLE)
      Ack_M422 : Bool;   // ACKNOWLEDGE M422-FIXTURE 1 AXIAL LOCATOR RETURN (READ-IN DISABLE)
      M423 : Bool;   // M423-FIXTURE 1 AXIAL LOCATOR RETURN
      Ack_M423 : Bool;   // ACKNOWLEDGE M423-FIXTURE 1 AXIAL LOCATOR RETURN
      M424 : Bool;   // M424-FIXTURE 1 AXIAL LOCATOR RELEASE PRESSURE (READ-IN DISABLE)
      Ack_M424 : Bool;   // ACKNOWLEDGE M424-FIXTURE 1 AXIAL LOCATOR RELEASE PRESSURE (READ-IN DISABLE)
      M425 : Bool;   // M425-FIXTURE 1 AXIAL LOCATOR LOW PRESSURE (READ-IN DISABLE)
      Ack_M425 : Bool;   // ACKNOWLEDGE M425-FIXTURE 1 AXIAL LOCATOR LOW PRESSURE (READ-IN DISABLE)
      M426 : Bool;   // M426-FIXTURE 1 AXIAL LOCATOR CARRIER ADVANCE (READ-IN DISABLE)
      Ack_M426 : Bool;   // ACKNOWLEDGE M426-FIXTURE 1 AXIAL LOCATOR CARRIER ADVANCE (READ-IN DISABLE)
      M427 : Bool;   // M427-FIXTURE 1 AXIAL LOCATOR CARRIER ADVANCE
      Ack_M427 : Bool;   // ACKNOWLEDGE M427-FIXTURE 1 AXIAL LOCATOR CARRIER ADVANCE
      M428 : Bool;   // M428-FIXTURE 1 AXIAL LOCATOR CARRIER RETURN (READ-IN DISABLE)
      Ack_M428 : Bool;   // ACKNOWLEDGE M428-FIXTURE 1 AXIAL LOCATOR CARRIER RETURN (READ-IN DISABLE)
      M429 : Bool;   // M429-FIXTURE 1 AXIAL LOCATOR CARRIER RETURN
      Ack_M429 : Bool;   // ACKNOWLEDGE M429-FIXTURE 1 AXIAL LOCATOR CARRIER RETURN
      M430 : Bool;   // M430-FIXTURE 1 AXIAL LOCATOR CARRIER RELEASE PRESSURE (READ-IN DISABLE)
      Ack_M430 : Bool;   // ACKNOWLEDGE M430-FIXTURE 1 AXIAL LOCATOR CARRIER RELEASE PRESSURE (READ-IN DISABLE)
      M431 : Bool;   // M431-FIXTURE 1 AXIAL LOCATOR CARRIER LOW PRESSURE (READ-IN DISABLE)
      Ack_M431 : Bool;   // ACKNOWLEDGE M431-FIXTURE 1 AXIAL LOCATOR CARRIER LOW PRESSURE (READ-IN DISABLE)
      M432 : Bool;   // M432-
      Ack_M432 : Bool;   // ACKNOWLEDGE M432-
      M433 : Bool;   // M433-
      Ack_M433 : Bool;   // ACKNOWLEDGE M433-
      M434 : Bool;   // M434-
      Ack_M434 : Bool;   // ACKNOWLEDGE M434-
      M435 : Bool;   // M435-
      Ack_M435 : Bool;   // ACKNOWLEDGE M435-
      M436 : Bool;   // M436-
      Ack_M436 : Bool;   // ACKNOWLEDGE M436-
      M437 : Bool;   // M437-
      Ack_M437 : Bool;   // ACKNOWLEDGE M437-
      M438 : Bool;   // M438-
      Ack_M438 : Bool;   // ACKNOWLEDGE M438-
      M439 : Bool;   // M439-
      Ack_M439 : Bool;   // ACKNOWLEDGE M439-
      M440 : Bool;   // M440-
      Ack_M440 : Bool;   // ACKNOWLEDGE M440-
      M441 : Bool;   // M441-
      Ack_M441 : Bool;   // ACKNOWLEDGE M441-
      M442 : Bool;   // M442-
      Ack_M442 : Bool;   // ACKNOWLEDGE M442-
      M443 : Bool;   // M443-
      Ack_M443 : Bool;   // ACKNOWLEDGE M443-
      M444 : Bool;   // M444-FIXTURE 1 RADIAL LOCATOR LOCATE (READ-IN DISABLE)
      Ack_M444 : Bool;   // ACKNOWLEDGE M444-FIXTURE 1 RADIAL LOCATOR LOCATE (READ-IN DISABLE)
      M445 : Bool;   // M445-FIXTURE 1 RADIAL LOCATOR LOCATE
      Ack_M445 : Bool;   // ACKNOWLEDGE M445-FIXTURE 1 RADIAL LOCATOR LOCATE
      M446 : Bool;   // M446-FIXTURE 1 RADIAL LOCATOR RETURN (READ-IN DISABLE)
      Ack_M446 : Bool;   // ACKNOWLEDGE M446-FIXTURE 1 RADIAL LOCATOR RETURN (READ-IN DISABLE)
      M447 : Bool;   // M447-FIXTURE 1 RADIAL LOCATOR RETURN
      Ack_M447 : Bool;   // ACKNOWLEDGE M447-FIXTURE 1 RADIAL LOCATOR RETURN
      M448 : Bool;   // M448-FIXTURE 1 RADIAL LOCATOR RELEASE PRESSURE (READ-IN DISABLE)
      Ack_M448 : Bool;   // ACKNOWLEDGE M448-FIXTURE 1 RADIAL LOCATOR RELEASE PRESSURE (READ-IN DISABLE)
      M449 : Bool;   // M449-FIXTURE 1 RADIAL LOCATOR LOW PRESSURE (READ-IN DISABLE)
      Ack_M449 : Bool;   // ACKNOWLEDGE M449-FIXTURE 1 RADIAL LOCATOR LOW PRESSURE (READ-IN DISABLE)
      M450 : Bool;   // M450-FIXTURE 1 RADIAL LOCATOR CARRIER ADVANCE (READ-IN DISABLE)
      Ack_M450 : Bool;   // ACKNOWLEDGE M450-FIXTURE 1 RADIAL LOCATOR CARRIER ADVANCE (READ-IN DISABLE)
      M451 : Bool;   // M451-FIXTURE 1 RADIAL LOCATOR CARRIER ADVANCE
      Ack_M451 : Bool;   // ACKNOWLEDGE M451-FIXTURE 1 RADIAL LOCATOR CARRIER ADVANCE
      M452 : Bool;   // M452-FIXTURE 1 RADIAL LOCATOR CARRIER RETURN (READ-IN DISABLE)
      Ack_M452 : Bool;   // ACKNOWLEDGE M452-FIXTURE 1 RADIAL LOCATOR CARRIER RETURN (READ-IN DISABLE)
      M453 : Bool;   // M453-FIXTURE 1 RADIAL LOCATOR CARRIER RETURN
      Ack_M453 : Bool;   // ACKNOWLEDGE M453-FIXTURE 1 RADIAL LOCATOR CARRIER RETURN
      M454 : Bool;   // M454-FIXTURE 1 RADIAL LOCATOR CARRIER RELEASE PRESSURE (READ-IN DISABLE)
      Ack_M454 : Bool;   // ACKNOWLEDGE M454-FIXTURE 1 RADIAL LOCATOR CARRIER RELEASE PRESSURE (READ-IN DISABLE)
      M455 : Bool;   // M455-FIXTURE 1 RADIAL LOCATOR CARRIER LOW PRESSURE (READ-IN DISABLE)
      Ack_M455 : Bool;   // ACKNOWLEDGE M455-FIXTURE 1 RADIAL LOCATOR CARRIER LOW PRESSURE (READ-IN DISABLE)
      M456 : Bool;   // M456-
      Ack_M456 : Bool;   // ACKNOWLEDGE M456-
      M457 : Bool;   // M457-
      Ack_M457 : Bool;   // ACKNOWLEDGE M457-
      M458 : Bool;   // M458-
      Ack_M458 : Bool;   // ACKNOWLEDGE M458-
      M459 : Bool;   // M459-
      Ack_M459 : Bool;   // ACKNOWLEDGE M459-
      M460 : Bool;   // M460-
      Ack_M460 : Bool;   // ACKNOWLEDGE M460-
      M461 : Bool;   // M461-
      Ack_M461 : Bool;   // ACKNOWLEDGE M461-
      M462 : Bool;   // M462-
      Ack_M462 : Bool;   // ACKNOWLEDGE M462-
      M463 : Bool;   // M463-
      Ack_M463 : Bool;   // ACKNOWLEDGE M463-
      M464 : Bool;   // M464-
      Ack_M464 : Bool;   // ACKNOWLEDGE M464-
      M465 : Bool;   // M465-
      Ack_M465 : Bool;   // ACKNOWLEDGE M465-
      M466 : Bool;   // M466-
      Ack_M466 : Bool;   // ACKNOWLEDGE M466-
      M467 : Bool;   // M467-
      Ack_M467 : Bool;   // ACKNOWLEDGE M467-
      M468 : Bool;   // M468-FIXTURE 1 CLAMPING FLANGE CLAMP (READ-IN DISABLE)
      Ack_M468 : Bool;   // ACKNOWLEDGE M468-FIXTURE 1 CLAMPING FLANGE CLAMP (READ-IN DISABLE)
      M469 : Bool;   // M469-FIXTURE 1 CLAMPING FLANGE CLAMP
      Ack_M469 : Bool;   // ACKNOWLEDGE M469-FIXTURE 1 CLAMPING FLANGE CLAMP
      M470 : Bool;   // M470-FIXTURE 1 CLAMPING FLANGE UNCLAMP (READ-IN DISABLE)
      Ack_M470 : Bool;   // ACKNOWLEDGE M470-FIXTURE 1 CLAMPING FLANGE UNCLAMP (READ-IN DISABLE)
      M471 : Bool;   // M471-FIXTURE 1 CLAMPING FLANGE UNCLAMP
      Ack_M471 : Bool;   // ACKNOWLEDGE M471-FIXTURE 1 CLAMPING FLANGE UNCLAMP
      M472 : Bool;   // M472-FIXTURE 1 CLAMPING FLANGE RELEASE PRESSURE (READ-IN DISABLE)
      Ack_M472 : Bool;   // ACKNOWLEDGE M472-FIXTURE 1 CLAMPING FLANGE RELEASE PRESSURE (READ-IN DISABLE)
      M473 : Bool;   // M473-FIXTURE 1 CLAMPING FLANGE LOW PRESSURE (READ-IN DISABLE)
      Ack_M473 : Bool;   // ACKNOWLEDGE M473-FIXTURE 1 CLAMPING FLANGE LOW PRESSURE (READ-IN DISABLE)
      M474 : Bool;   // M474-
      Ack_M474 : Bool;   // ACKNOWLEDGE M474-
      M475 : Bool;   // M475-
      Ack_M475 : Bool;   // ACKNOWLEDGE M475-
      M476 : Bool;   // M476-
      Ack_M476 : Bool;   // ACKNOWLEDGE M476-
      M477 : Bool;   // M477-
      Ack_M477 : Bool;   // ACKNOWLEDGE M477-
      M478 : Bool;   // M478-
      Ack_M478 : Bool;   // ACKNOWLEDGE M478-
      M479 : Bool;   // M479-
      Ack_M479 : Bool;   // ACKNOWLEDGE M479-
      M480 : Bool;   // M480-
      Ack_M480 : Bool;   // ACKNOWLEDGE M480-
      M481 : Bool;   // M481-
      Ack_M481 : Bool;   // ACKNOWLEDGE M481-
      M482 : Bool;   // M482-
      Ack_M482 : Bool;   // ACKNOWLEDGE M482-
      M483 : Bool;   // M483-
      Ack_M483 : Bool;   // ACKNOWLEDGE M483-
      M484 : Bool;   // M484-
      Ack_M484 : Bool;   // ACKNOWLEDGE M484-
      M485 : Bool;   // M485-
      Ack_M485 : Bool;   // ACKNOWLEDGE M485-
      M486 : Bool;   // M486-FIXTURE 1 TAILSTOCK ADVANCE (READ-IN DISABLE)
      Ack_M486 : Bool;   // ACKNOWLEDGE M486-FIXTURE 1 TAILSTOCK ADVANCE (READ-IN DISABLE)
      M487 : Bool;   // M487-FIXTURE 1 TAILSTOCK ADVANCE
      Ack_M487 : Bool;   // ACKNOWLEDGE M487-FIXTURE 1 TAILSTOCK ADVANCE
      M488 : Bool;   // M488-FIXTURE 1 TAILSTOCK RETURN (READ-IN DISABLE)
      Ack_M488 : Bool;   // ACKNOWLEDGE M488-FIXTURE 1 TAILSTOCK RETURN (READ-IN DISABLE)
      M489 : Bool;   // M489-FIXTURE 1 TAILSTOCK RETURN
      Ack_M489 : Bool;   // ACKNOWLEDGE M489-FIXTURE 1 TAILSTOCK RETURN
      M490 : Bool;   // M490-FIXTURE 1 TAILSTOCK RELEASE PRESSURE (READ-IN DISABLE)
      Ack_M490 : Bool;   // ACKNOWLEDGE M490-FIXTURE 1 TAILSTOCK RELEASE PRESSURE (READ-IN DISABLE)
      M491 : Bool;   // M491-FIXTURE 1 TAILSTOCK LOW PRESSURE (READ-IN DISABLE)
      Ack_M491 : Bool;   // ACKNOWLEDGE M491-FIXTURE 1 TAILSTOCK LOW PRESSURE (READ-IN DISABLE)
      M492 : Bool;   // M492-
      Ack_M492 : Bool;   // ACKNOWLEDGE M492-
      M493 : Bool;   // M493-
      Ack_M493 : Bool;   // ACKNOWLEDGE M493-
      M494 : Bool;   // M494-
      Ack_M494 : Bool;   // ACKNOWLEDGE M494-
      M495 : Bool;   // M495-
      Ack_M495 : Bool;   // ACKNOWLEDGE M495-
      M496 : Bool;   // M496-
      Ack_M496 : Bool;   // ACKNOWLEDGE M496-
      M497 : Bool;   // M497-
      Ack_M497 : Bool;   // ACKNOWLEDGE M497-
      M498 : Bool;   // M498-FIXTURE 1 SHIFTING DEVICE LOCATE (READ-IN DISABLE)
      Ack_M498 : Bool;   // ACKNOWLEDGE M498-FIXTURE 1 SHIFTING DEVICE LOCATE (READ-IN DISABLE)
      M499 : Bool;   // M499-FIXTURE 1 SHIFTING DEVICE LOCATE
      Ack_M499 : Bool;   // ACKNOWLEDGE M499-FIXTURE 1 SHIFTING DEVICE LOCATE
      M500 : Bool;   // M500-FIXTURE 1 SHIFTING DEVICE RETURN (READ-IN DISABLE)
      Ack_M500 : Bool;   // ACKNOWLEDGE M500-FIXTURE 1 SHIFTING DEVICE RETURN (READ-IN DISABLE)
      M501 : Bool;   // M501-FIXTURE 1 SHIFTING DEVICE RETURN
      Ack_M501 : Bool;   // ACKNOWLEDGE M501-FIXTURE 1 SHIFTING DEVICE RETURN
      M502 : Bool;   // M502-FIXTURE 1 SHIFTING DEVICE RELEASE PRESSURE (READ-IN DISABLE)
      Ack_M502 : Bool;   // ACKNOWLEDGE M502-FIXTURE 1 SHIFTING DEVICE RELEASE PRESSURE (READ-IN DISABLE)
      M503 : Bool;   // M503-FIXTURE 1 SHIFTING DEVICE LOW PRESSURE (READ-IN DISABLE)
      Ack_M503 : Bool;   // ACKNOWLEDGE M503-FIXTURE 1 SHIFTING DEVICE LOW PRESSURE (READ-IN DISABLE)
      M504 : Bool;   // M504-FIXTURE 1 BLOCKING DEVICE BLOCK (READ-IN DISABLE)
      Ack_M504 : Bool;   // ACKNOWLEDGE M504-FIXTURE 1 BLOCKING DEVICE BLOCK (READ-IN DISABLE)
      M505 : Bool;   // M505-FIXTURE 1 BLOCKING DEVICE BLOCK
      Ack_M505 : Bool;   // ACKNOWLEDGE M505-FIXTURE 1 BLOCKING DEVICE BLOCK
      M506 : Bool;   // M506-FIXTURE 1 BLOCKING DEVICE UNBLOCK (READ-IN DISABLE)
      Ack_M506 : Bool;   // ACKNOWLEDGE M506-FIXTURE 1 BLOCKING DEVICE UNBLOCK (READ-IN DISABLE)
      M507 : Bool;   // M507-FIXTURE 1 BLOCKING DEVICE UNBLOCK
      Ack_M507 : Bool;   // ACKNOWLEDGE M507-FIXTURE 1 BLOCKING DEVICE UNBLOCK
      M508 : Bool;   // M508-FIXTURE 1 BLOCKING DEVICE RELEASE PRESSURE (READ-IN DISABLE)
      Ack_M508 : Bool;   // ACKNOWLEDGE M508-FIXTURE 1 BLOCKING DEVICE RELEASE PRESSURE (READ-IN DISABLE)
      M509 : Bool;   // M509-FIXTURE 1 BLOCKING DEVICE LOW PRESSURE (READ-IN DISABLE)
      Ack_M509 : Bool;   // ACKNOWLEDGE M509-FIXTURE 1 BLOCKING DEVICE LOW PRESSURE (READ-IN DISABLE)
      M510 : Bool;   // M510-FIXTURE 1 VIBRATION DAMPER CLAMP (READ-IN DISABLE)
      Ack_M510 : Bool;   // ACKNOWLEDGE M510-FIXTURE 1 VIBRATION DAMPER CLAMP (READ-IN DISABLE)
      M511 : Bool;   // M511-FIXTURE 1 VIBRATION DAMPER CLAMP
      Ack_M511 : Bool;   // ACKNOWLEDGE M511-FIXTURE 1 VIBRATION DAMPER CLAMP
      M512 : Bool;   // M512-FIXTURE 1 VIBRATION DAMPER UNCLAMP (READ-IN DISABLE)
      Ack_M512 : Bool;   // ACKNOWLEDGE M512-FIXTURE 1 VIBRATION DAMPER UNCLAMP (READ-IN DISABLE)
      M513 : Bool;   // M513-FIXTURE 1 VIBRATION DAMPER UNCLAMP
      Ack_M513 : Bool;   // ACKNOWLEDGE M513-FIXTURE 1 VIBRATION DAMPER UNCLAMP
      M514 : Bool;   // M514-FIXTURE 1 VIBRATION DAMPER RELEASE PRESSURE (READ-IN DISABLE)
      Ack_M514 : Bool;   // ACKNOWLEDGE M514-FIXTURE 1 VIBRATION DAMPER RELEASE PRESSURE (READ-IN DISABLE)
      M515 : Bool;   // M515-FIXTURE 1 VIBRATION DAMPER LOW PRESSURE (READ-IN DISABLE)
      Ack_M515 : Bool;   // ACKNOWLEDGE M515-FIXTURE 1 VIBRATION DAMPER LOW PRESSURE (READ-IN DISABLE)
      M516 : Bool;   // M516-
      Ack_M516 : Bool;   // ACKNOWLEDGE M516-
      M517 : Bool;   // M517-
      Ack_M517 : Bool;   // ACKNOWLEDGE M517-
      M518 : Bool;   // M518-
      Ack_M518 : Bool;   // ACKNOWLEDGE M518-
      M519 : Bool;   // M519-
      Ack_M519 : Bool;   // ACKNOWLEDGE M519-
      M520 : Bool;   // M520-
      Ack_M520 : Bool;   // ACKNOWLEDGE M520-
      M521 : Bool;   // M521-
      Ack_M521 : Bool;   // ACKNOWLEDGE M521-
      M522 : Bool;   // M522-
      Ack_M522 : Bool;   // ACKNOWLEDGE M522-
      M523 : Bool;   // M523-
      Ack_M523 : Bool;   // ACKNOWLEDGE M523-
      M524 : Bool;   // M524-
      Ack_M524 : Bool;   // ACKNOWLEDGE M524-
      M525 : Bool;   // M525-
      Ack_M525 : Bool;   // ACKNOWLEDGE M525-
      M526 : Bool;   // M526-
      Ack_M526 : Bool;   // ACKNOWLEDGE M526-
      M527 : Bool;   // M527-
      Ack_M527 : Bool;   // ACKNOWLEDGE M527-
      M528 : Bool;   // M528-FIXTURE 1 JAW CHUCK CLAMP (READ-IN DISABLE)
      Ack_M528 : Bool;   // ACKNOWLEDGE M528-FIXTURE 1 JAW CHUCK CLAMP (READ-IN DISABLE)
      M529 : Bool;   // M529-FIXTURE 1 JAW CHUCK CLAMP
      Ack_M529 : Bool;   // ACKNOWLEDGE M529-FIXTURE 1 JAW CHUCK CLAMP
      M530 : Bool;   // M530-FIXTURE 1 JAW CHUCK UNCLAMP (READ-IN DISABLE)
      Ack_M530 : Bool;   // ACKNOWLEDGE M530-FIXTURE 1 JAW CHUCK UNCLAMP (READ-IN DISABLE)
      M531 : Bool;   // M531-FIXTURE 1 JAW CHUCK UNCLAMP
      Ack_M531 : Bool;   // ACKNOWLEDGE M531-FIXTURE 1 JAW CHUCK UNCLAMP
      M532 : Bool;   // M532-FIXTURE 1 JAW CHUCK RELEASE PRESSURE (READ-IN DISABLE)
      Ack_M532 : Bool;   // ACKNOWLEDGE M532-FIXTURE 1 JAW CHUCK RELEASE PRESSURE (READ-IN DISABLE)
      M533 : Bool;   // M533-FIXTURE 1 JAW CHUCK LOW CLAMP (READ-IN DISABLE)
      Ack_M533 : Bool;   // ACKNOWLEDGE M533-FIXTURE 1 JAW CHUCK LOW CLAMP (READ-IN DISABLE)
      M534 : Bool;   // M534-
      Ack_M534 : Bool;   // ACKNOWLEDGE M534-
      M535 : Bool;   // M535-
      Ack_M535 : Bool;   // ACKNOWLEDGE M535-
      M536 : Bool;   // M536-
      Ack_M536 : Bool;   // ACKNOWLEDGE M536-
      M537 : Bool;   // M537-
      Ack_M537 : Bool;   // ACKNOWLEDGE M537-
      M538 : Bool;   // M538-
      Ack_M538 : Bool;   // ACKNOWLEDGE M538-
      M539 : Bool;   // M539-
      Ack_M539 : Bool;   // ACKNOWLEDGE M539-
      M540 : Bool;   // M540-
      Ack_M540 : Bool;   // ACKNOWLEDGE M540-
      M541 : Bool;   // M541-
      Ack_M541 : Bool;   // ACKNOWLEDGE M541-
      M542 : Bool;   // M542-
      Ack_M542 : Bool;   // ACKNOWLEDGE M542-
      M543 : Bool;   // M543-
      Ack_M543 : Bool;   // ACKNOWLEDGE M543-
      M544 : Bool;   // M544-
      Ack_M544 : Bool;   // ACKNOWLEDGE M544-
      M545 : Bool;   // M545-
      Ack_M545 : Bool;   // ACKNOWLEDGE M545-
      M546 : Bool;   // M546-FIXTURE 1 CENTRAL JAW CHUCK CLAMP (READ-IN DISABLE)
      Ack_M546 : Bool;   // ACKNOWLEDGE M546-FIXTURE 1 CENTRAL JAW CHUCK CLAMP (READ-IN DISABLE)
      M547 : Bool;   // M547-FIXTURE 1 CENTRAL JAW CHUCK CLAMP
      Ack_M547 : Bool;   // ACKNOWLEDGE M547-FIXTURE 1 CENTRAL JAW CHUCK CLAMP
      M548 : Bool;   // M548-FIXTURE 1 CENTRAL JAW CHUCK UNCLAMP (READ-IN DISABLE)
      Ack_M548 : Bool;   // ACKNOWLEDGE M548-FIXTURE 1 CENTRAL JAW CHUCK UNCLAMP (READ-IN DISABLE)
      M549 : Bool;   // M549-FIXTURE 1 CENTRAL JAW CHUCK UNCLAMP
      Ack_M549 : Bool;   // ACKNOWLEDGE M549-FIXTURE 1 CENTRAL JAW CHUCK UNCLAMP
      M550 : Bool;   // M550-FIXTURE 1 CENTRAL JAW CHUCK RELEASE PRESSURE (READ-IN DISABLE)
      Ack_M550 : Bool;   // ACKNOWLEDGE M550-FIXTURE 1 CENTRAL JAW CHUCK RELEASE PRESSURE (READ-IN DISABLE)
      M551 : Bool;   // M551-FIXTURE 1 CENTRAL JAW CHUCK LOW CLAMP (READ-IN DISABLE)
      Ack_M551 : Bool;   // ACKNOWLEDGE M551-FIXTURE 1 CENTRAL JAW CHUCK LOW CLAMP (READ-IN DISABLE)
      M552 : Bool;   // M552-
      Ack_M552 : Bool;   // ACKNOWLEDGE M552-
      M553 : Bool;   // M553-
      Ack_M553 : Bool;   // ACKNOWLEDGE M553-
      M554 : Bool;   // M554-
      Ack_M554 : Bool;   // ACKNOWLEDGE M554-
      M555 : Bool;   // M555-
      Ack_M555 : Bool;   // ACKNOWLEDGE M555-
      M556 : Bool;   // M556-
      Ack_M556 : Bool;   // ACKNOWLEDGE M556-
      M557 : Bool;   // M557-
      Ack_M557 : Bool;   // ACKNOWLEDGE M557-
      M558 : Bool;   // M558-
      Ack_M558 : Bool;   // ACKNOWLEDGE M558-
      M559 : Bool;   // M559-
      Ack_M559 : Bool;   // ACKNOWLEDGE M559-
      M560 : Bool;   // M560-
      Ack_M560 : Bool;   // ACKNOWLEDGE M560-
      M561 : Bool;   // M561-
      Ack_M561 : Bool;   // ACKNOWLEDGE M561-
      M562 : Bool;   // M562-
      Ack_M562 : Bool;   // ACKNOWLEDGE M562-
      M563 : Bool;   // M563-
      Ack_M563 : Bool;   // ACKNOWLEDGE M563-
      M564 : Bool;   // M564-FIXTURE 1 JAW CHUCK B CLAMP (READ-IN DISABLE)
      Ack_M564 : Bool;   // ACKNOWLEDGE M564-FIXTURE 1 JAW CHUCK B CLAMP (READ-IN DISABLE)
      M565 : Bool;   // M565-FIXTURE 1 JAW CHUCK B CLAMP
      Ack_M565 : Bool;   // ACKNOWLEDGE M565-FIXTURE 1 JAW CHUCK B CLAMP
      M566 : Bool;   // M566-FIXTURE 1 JAW CHUCK B UNCLAMP (READ-IN DISABLE)
      Ack_M566 : Bool;   // ACKNOWLEDGE M566-FIXTURE 1 JAW CHUCK B UNCLAMP (READ-IN DISABLE)
      M567 : Bool;   // M567-FIXTURE 1 JAW CHUCK B UNCLAMP
      Ack_M567 : Bool;   // ACKNOWLEDGE M567-FIXTURE 1 JAW CHUCK B UNCLAMP
      M568 : Bool;   // M568-FIXTURE 1 JAW CHUCK B RELEASE PRESSURE (READ-IN DISABLE)
      Ack_M568 : Bool;   // ACKNOWLEDGE M568-FIXTURE 1 JAW CHUCK B RELEASE PRESSURE (READ-IN DISABLE)
      M569 : Bool;   // M569-FIXTURE 1 JAW CHUCK B LOW PRESSURE (READ-IN DISABLE)
      Ack_M569 : Bool;   // ACKNOWLEDGE M569-FIXTURE 1 JAW CHUCK B LOW PRESSURE (READ-IN DISABLE)
      M570 : Bool;   // M570-FIXTURE 1 ROTARY JAW CHUCK CLAMP (READ-IN DISABLE)
      Ack_M570 : Bool;   // ACKNOWLEDGE M570-FIXTURE 1 ROTARY JAW CHUCK CLAMP (READ-IN DISABLE)
      M571 : Bool;   // M571-FIXTURE 1 ROTARY JAW CHUCK CLAMP
      Ack_M571 : Bool;   // ACKNOWLEDGE M571-FIXTURE 1 ROTARY JAW CHUCK CLAMP
      M572 : Bool;   // M572-FIXTURE 1 ROTARY JAW CHUCK UNCLAMP (READ-IN DISABLE)
      Ack_M572 : Bool;   // ACKNOWLEDGE M572-FIXTURE 1 ROTARY JAW CHUCK UNCLAMP (READ-IN DISABLE)
      M573 : Bool;   // M573-FIXTURE 1 ROTARY JAW CHUCK UNCLAMP
      Ack_M573 : Bool;   // ACKNOWLEDGE M573-FIXTURE 1 ROTARY JAW CHUCK UNCLAMP
      M574 : Bool;   // M574-FIXTURE 1 ROTARY JAW CHUCK RELEASE PRESSURE (READ-IN DISABLE)
      Ack_M574 : Bool;   // ACKNOWLEDGE M574-FIXTURE 1 ROTARY JAW CHUCK RELEASE PRESSURE (READ-IN DISABLE)
      M575 : Bool;   // M575-FIXTURE 1 ROTARY JAW CHUCK LOW PRESSURE (READ-IN DISABLE)
      Ack_M575 : Bool;   // ACKNOWLEDGE M575-FIXTURE 1 ROTARY JAW CHUCK LOW PRESSURE (READ-IN DISABLE)
      M576 : Bool;   // M576-
      Ack_M576 : Bool;   // ACKNOWLEDGE M576-
      M577 : Bool;   // M577-
      Ack_M577 : Bool;   // ACKNOWLEDGE M577-
      M578 : Bool;   // M578-
      Ack_M578 : Bool;   // ACKNOWLEDGE M578-
      M579 : Bool;   // M579-
      Ack_M579 : Bool;   // ACKNOWLEDGE M579-
      M580 : Bool;   // M580-
      Ack_M580 : Bool;   // ACKNOWLEDGE M580-
      M581 : Bool;   // M581-
      Ack_M581 : Bool;   // ACKNOWLEDGE M581-
      M582 : Bool;   // M582-
      Ack_M582 : Bool;   // ACKNOWLEDGE M582-
      M583 : Bool;   // M583-
      Ack_M583 : Bool;   // ACKNOWLEDGE M583-
      M584 : Bool;   // M584-
      Ack_M584 : Bool;   // ACKNOWLEDGE M584-
      M585 : Bool;   // M585-
      Ack_M585 : Bool;   // ACKNOWLEDGE M585-
      M586 : Bool;   // M586-
      Ack_M586 : Bool;   // ACKNOWLEDGE M586-
      M587 : Bool;   // M587-
      Ack_M587 : Bool;   // ACKNOWLEDGE M587-
      M588 : Bool;   // M588-FIXTURE 1 REMOVABLE STOP ADVANCE (READ-IN DISABLE)
      Ack_M588 : Bool;   // ACKNOWLEDGE M588-FIXTURE 1 REMOVABLE STOP ADVANCE (READ-IN DISABLE)
      M589 : Bool;   // M589-FIXTURE 1 REMOVABLE STOP ADVANCE
      Ack_M589 : Bool;   // ACKNOWLEDGE M589-FIXTURE 1 REMOVABLE STOP ADVANCE
      M590 : Bool;   // M590-FIXTURE 1 REMOVABLE STOP RETURN (READ-IN DISABLE)
      Ack_M590 : Bool;   // ACKNOWLEDGE M590-FIXTURE 1 REMOVABLE STOP RETURN (READ-IN DISABLE)
      M591 : Bool;   // M591-FIXTURE 1 REMOVABLE STOP RETURN
      Ack_M591 : Bool;   // ACKNOWLEDGE M591-FIXTURE 1 REMOVABLE STOP RETURN
      M592 : Bool;   // M592-FIXTURE 1 REMOVABLE STOP RELEASE PRESSURE (READ-IN DISABLE)
      Ack_M592 : Bool;   // ACKNOWLEDGE M592-FIXTURE 1 REMOVABLE STOP RELEASE PRESSURE (READ-IN DISABLE)
      M593 : Bool;   // M593-FIXTURE 1 REMOVABLE STOP LOW PRESSURE (READ-IN DISABLE)
      Ack_M593 : Bool;   // ACKNOWLEDGE M593-FIXTURE 1 REMOVABLE STOP LOW PRESSURE (READ-IN DISABLE)
      M594 : Bool;   // M594-
      Ack_M594 : Bool;   // ACKNOWLEDGE M594-
      M595 : Bool;   // M595-
      Ack_M595 : Bool;   // ACKNOWLEDGE M595-
      M596 : Bool;   // M596-
      Ack_M596 : Bool;   // ACKNOWLEDGE M596-
      M597 : Bool;   // M597-
      Ack_M597 : Bool;   // ACKNOWLEDGE M597-
      M598 : Bool;   // M598-
      Ack_M598 : Bool;   // ACKNOWLEDGE M598-
      M599 : Bool;   // M599-
      Ack_M599 : Bool;   // ACKNOWLEDGE M599-
      M600 : Bool;   // M600-
      Ack_M600 : Bool;   // ACKNOWLEDGE M600-
      M601 : Bool;   // M601-
      Ack_M601 : Bool;   // ACKNOWLEDGE M601-
      M602 : Bool;   // M602-
      Ack_M602 : Bool;   // ACKNOWLEDGE M602-
      M603 : Bool;   // M603-
      Ack_M603 : Bool;   // ACKNOWLEDGE M603-
      M604 : Bool;   // M604-
      Ack_M604 : Bool;   // ACKNOWLEDGE M604-
      M605 : Bool;   // M605-
      Ack_M605 : Bool;   // ACKNOWLEDGE M605-
      M606 : Bool;   // M606-
      Ack_M606 : Bool;   // ACKNOWLEDGE M606-
      M607 : Bool;   // M607-
      Ack_M607 : Bool;   // ACKNOWLEDGE M607-
      M608 : Bool;   // M608-
      Ack_M608 : Bool;   // ACKNOWLEDGE M608-
      M609 : Bool;   // M609-
      Ack_M609 : Bool;   // ACKNOWLEDGE M609-
      M610 : Bool;   // M610-
      Ack_M610 : Bool;   // ACKNOWLEDGE M610-
      M611 : Bool;   // M611-
      Ack_M611 : Bool;   // ACKNOWLEDGE M611-
      M612 : Bool;   // M612-
      Ack_M612 : Bool;   // ACKNOWLEDGE M612-
      M613 : Bool;   // M613-
      Ack_M613 : Bool;   // ACKNOWLEDGE M613-
      M614 : Bool;   // M614-
      Ack_M614 : Bool;   // ACKNOWLEDGE M614-
      M615 : Bool;   // M615-
      Ack_M615 : Bool;   // ACKNOWLEDGE M615-
      M616 : Bool;   // M616-
      Ack_M616 : Bool;   // ACKNOWLEDGE M616-
      M617 : Bool;   // M617-
      Ack_M617 : Bool;   // ACKNOWLEDGE M617-
      M618 : Bool;   // M618-
      Ack_M618 : Bool;   // ACKNOWLEDGE M618-
      M619 : Bool;   // M619-
      Ack_M619 : Bool;   // ACKNOWLEDGE M619-
      M620 : Bool;   // M620-
      Ack_M620 : Bool;   // ACKNOWLEDGE M620-
      M621 : Bool;   // M621-
      Ack_M621 : Bool;   // ACKNOWLEDGE M621-
      M622 : Bool;   // M622-
      Ack_M622 : Bool;   // ACKNOWLEDGE M622-
      M623 : Bool;   // M623-
      Ack_M623 : Bool;   // ACKNOWLEDGE M623-
      M624 : Bool;   // M624-
      Ack_M624 : Bool;   // ACKNOWLEDGE M624-
      M625 : Bool;   // M625-
      Ack_M625 : Bool;   // ACKNOWLEDGE M625-
      M626 : Bool;   // M626-
      Ack_M626 : Bool;   // ACKNOWLEDGE M626-
      M627 : Bool;   // M627-
      Ack_M627 : Bool;   // ACKNOWLEDGE M627-
      M628 : Bool;   // M628-
      Ack_M628 : Bool;   // ACKNOWLEDGE M628-
      M629 : Bool;   // M629-
      Ack_M629 : Bool;   // ACKNOWLEDGE M629-
      M630 : Bool;   // M630-
      Ack_M630 : Bool;   // ACKNOWLEDGE M630-
      M631 : Bool;   // M631-
      Ack_M631 : Bool;   // ACKNOWLEDGE M631-
      M632 : Bool;   // M632-
      Ack_M632 : Bool;   // ACKNOWLEDGE M632-
      M633 : Bool;   // M633-
      Ack_M633 : Bool;   // ACKNOWLEDGE M633-
      M634 : Bool;   // M634-
      Ack_M634 : Bool;   // ACKNOWLEDGE M634-
      M635 : Bool;   // M635-
      Ack_M635 : Bool;   // ACKNOWLEDGE M635-
      M636 : Bool;   // M636-
      Ack_M636 : Bool;   // ACKNOWLEDGE M636-
      M637 : Bool;   // M637-
      Ack_M637 : Bool;   // ACKNOWLEDGE M637-
      M638 : Bool;   // M638-
      Ack_M638 : Bool;   // ACKNOWLEDGE M638-
      M639 : Bool;   // M639-
      Ack_M639 : Bool;   // ACKNOWLEDGE M639-
      M640 : Bool;   // M640-
      Ack_M640 : Bool;   // ACKNOWLEDGE M640-
      M641 : Bool;   // M641-
      Ack_M641 : Bool;   // ACKNOWLEDGE M641-
      M642 : Bool;   // M642-
      Ack_M642 : Bool;   // ACKNOWLEDGE M642-
      M643 : Bool;   // M643-
      Ack_M643 : Bool;   // ACKNOWLEDGE M643-
      M644 : Bool;   // M644-
      Ack_M644 : Bool;   // ACKNOWLEDGE M644-
      M645 : Bool;   // M645-
      Ack_M645 : Bool;   // ACKNOWLEDGE M645-
      M646 : Bool;   // M646-
      Ack_M646 : Bool;   // ACKNOWLEDGE M646-
      M647 : Bool;   // M647-
      Ack_M647 : Bool;   // ACKNOWLEDGE M647-
      M648 : Bool;   // M648-
      Ack_M648 : Bool;   // ACKNOWLEDGE M648-
      M649 : Bool;   // M649-
      Ack_M649 : Bool;   // ACKNOWLEDGE M649-
      M650 : Bool;   // M650-
      Ack_M650 : Bool;   // ACKNOWLEDGE M650-
      M651 : Bool;   // M651-
      Ack_M651 : Bool;   // ACKNOWLEDGE M651-
      M652 : Bool;   // M652-
      Ack_M652 : Bool;   // ACKNOWLEDGE M652-
      M653 : Bool;   // M653-
      Ack_M653 : Bool;   // ACKNOWLEDGE M653-
      M654 : Bool;   // M654-
      Ack_M654 : Bool;   // ACKNOWLEDGE M654-
      M655 : Bool;   // M655-
      Ack_M655 : Bool;   // ACKNOWLEDGE M655-
      M656 : Bool;   // M656-
      Ack_M656 : Bool;   // ACKNOWLEDGE M656-
      M657 : Bool;   // M657-
      Ack_M657 : Bool;   // ACKNOWLEDGE M657-
      M658 : Bool;   // M658-
      Ack_M658 : Bool;   // ACKNOWLEDGE M658-
      M659 : Bool;   // M659-
      Ack_M659 : Bool;   // ACKNOWLEDGE M659-
      M660 : Bool;   // M660-
      Ack_M660 : Bool;   // ACKNOWLEDGE M660-
      M661 : Bool;   // M661-
      Ack_M661 : Bool;   // ACKNOWLEDGE M661-
      M662 : Bool;   // M662-
      Ack_M662 : Bool;   // ACKNOWLEDGE M662-
      M663 : Bool;   // M663-
      Ack_M663 : Bool;   // ACKNOWLEDGE M663-
      M664 : Bool;   // M664-
      Ack_M664 : Bool;   // ACKNOWLEDGE M664-
      M665 : Bool;   // M665-
      Ack_M665 : Bool;   // ACKNOWLEDGE M665-
      M666 : Bool;   // M666-
      Ack_M666 : Bool;   // ACKNOWLEDGE M666-
      M667 : Bool;   // M667-
      Ack_M667 : Bool;   // ACKNOWLEDGE M667-
      M668 : Bool;   // M668-
      Ack_M668 : Bool;   // ACKNOWLEDGE M668-
      M669 : Bool;   // M669-
      Ack_M669 : Bool;   // ACKNOWLEDGE M669-
      M670 : Bool;   // M670-
      Ack_M670 : Bool;   // ACKNOWLEDGE M670-
      M671 : Bool;   // M671-
      Ack_M671 : Bool;   // ACKNOWLEDGE M671-
      M672 : Bool;   // M672-
      Ack_M672 : Bool;   // ACKNOWLEDGE M672-
      M673 : Bool;   // M673-
      Ack_M673 : Bool;   // ACKNOWLEDGE M673-
      M674 : Bool;   // M674-
      Ack_M674 : Bool;   // ACKNOWLEDGE M674-
      M675 : Bool;   // M675-
      Ack_M675 : Bool;   // ACKNOWLEDGE M675-
      M676 : Bool;   // M676-
      Ack_M676 : Bool;   // ACKNOWLEDGE M676-
      M677 : Bool;   // M677-
      Ack_M677 : Bool;   // ACKNOWLEDGE M677-
      M678 : Bool;   // M678-
      Ack_M678 : Bool;   // ACKNOWLEDGE M678-
      M679 : Bool;   // M679-
      Ack_M679 : Bool;   // ACKNOWLEDGE M679-
      M680 : Bool;   // M680-
      Ack_M680 : Bool;   // ACKNOWLEDGE M680-
      M681 : Bool;   // M681-
      Ack_M681 : Bool;   // ACKNOWLEDGE M681-
      M682 : Bool;   // M682-
      Ack_M682 : Bool;   // ACKNOWLEDGE M682-
      M683 : Bool;   // M683-
      Ack_M683 : Bool;   // ACKNOWLEDGE M683-
      M684 : Bool;   // M684-
      Ack_M684 : Bool;   // ACKNOWLEDGE M684-
      M685 : Bool;   // M685-
      Ack_M685 : Bool;   // ACKNOWLEDGE M685-
      M686 : Bool;   // M686-
      Ack_M686 : Bool;   // ACKNOWLEDGE M686-
      M687 : Bool;   // M687-
      Ack_M687 : Bool;   // ACKNOWLEDGE M687-
      M688 : Bool;   // M688-
      Ack_M688 : Bool;   // ACKNOWLEDGE M688-
      M689 : Bool;   // M689-
      Ack_M689 : Bool;   // ACKNOWLEDGE M689-
      M690 : Bool;   // M690-
      Ack_M690 : Bool;   // ACKNOWLEDGE M690-
      M691 : Bool;   // M691-
      Ack_M691 : Bool;   // ACKNOWLEDGE M691-
      M692 : Bool;   // M692-
      Ack_M692 : Bool;   // ACKNOWLEDGE M692-
      M693 : Bool;   // M693-
      Ack_M693 : Bool;   // ACKNOWLEDGE M693-
      M694 : Bool;   // M694-
      Ack_M694 : Bool;   // ACKNOWLEDGE M694-
      M695 : Bool;   // M695-
      Ack_M695 : Bool;   // ACKNOWLEDGE M695-
      M696 : Bool;   // M696-
      Ack_M696 : Bool;   // ACKNOWLEDGE M696-
      M697 : Bool;   // M697-
      Ack_M697 : Bool;   // ACKNOWLEDGE M697-
      M698 : Bool;   // M698-
      Ack_M698 : Bool;   // ACKNOWLEDGE M698-
      M699 : Bool;   // M699-
      Ack_M699 : Bool;   // ACKNOWLEDGE M699-
      M700 : Bool;   // M700-FIXTURE 2 CLAMP SEQUENCE (READ-IN DISABLE)
      Ack_M700 : Bool;   // ACKNOWLEDGE M700-FIXTURE 2 CLAMP SEQUENCE (READ-IN DISABLE)
      M701 : Bool;   // M701-FIXTURE 2 CLAMP SEQUENCE
      Ack_M701 : Bool;   // ACKNOWLEDGE M701-FIXTURE 2 CLAMP SEQUENCE
      M702 : Bool;   // M702-FIXTURE 2 UNCLAMP SEQUENCE (READ-IN DISABLE)
      Ack_M702 : Bool;   // ACKNOWLEDGE M702-FIXTURE 2 UNCLAMP SEQUENCE (READ-IN DISABLE)
      M703 : Bool;   // M703-FIXTURE 2 UNCLAMP SEQUENCE
      Ack_M703 : Bool;   // ACKNOWLEDGE M703-FIXTURE 2 UNCLAMP SEQUENCE
      M704 : Bool;   // M704-FIXTURE 2 VERIFY PART AND TOOL IS CLAMPED DURING MACHINING (WHEN TRUE DO). TOGGLED
      Ack_M704 : Bool;   // ACKNOWLEDGE M704-FIXTURE 2 VERIFY PART AND TOOL IS CLAMPED DURING MACHINING (WHEN TRUE DO). TOGGLED
      M705 : Bool;   // M705-FIXTURE 2 VERIFY PART AND TOOL IS CLAMPED LOW PRESSURE DURING MACHINING (WHEN TRUE DO). TOGGLED
      Ack_M705 : Bool;   // ACKNOWLEDGE M705-FIXTURE 2 VERIFY PART AND TOOL IS CLAMPED LOW PRESSURE DURING MACHINING (WHEN TRUE DO). TOGGLED
      M706 : Bool;   // M706-FIXTURE 2 VERIFY PARTS ARE UNCLAMPED PARTS LOADING (WHEN TRUE DO). TOGGLED
      Ack_M706 : Bool;   // ACKNOWLEDGE M706-FIXTURE 2 VERIFY PARTS ARE UNCLAMPED PARTS LOADING (WHEN TRUE DO). TOGGLED
      M707 : Bool;   // M707-FIXTURE 2 VERIFY FIXTURE REMAINS CLAMPED
      Ack_M707 : Bool;   // ACKNOWLEDGE M707-FIXTURE 2 VERIFY FIXTURE REMAINS CLAMPED
      M708 : Bool;   // M708-
      Ack_M708 : Bool;   // ACKNOWLEDGE M708-
      M709 : Bool;   // M709-
      Ack_M709 : Bool;   // ACKNOWLEDGE M709-
      M710 : Bool;   // M710-
      Ack_M710 : Bool;   // ACKNOWLEDGE M710-
      M711 : Bool;   // M711-
      Ack_M711 : Bool;   // ACKNOWLEDGE M711-
      M712 : Bool;   // M712-
      Ack_M712 : Bool;   // ACKNOWLEDGE M712-
      M713 : Bool;   // M713-
      Ack_M713 : Bool;   // ACKNOWLEDGE M713-
      M714 : Bool;   // M714-
      Ack_M714 : Bool;   // ACKNOWLEDGE M714-
      M715 : Bool;   // M715-
      Ack_M715 : Bool;   // ACKNOWLEDGE M715-
      M716 : Bool;   // M716-
      Ack_M716 : Bool;   // ACKNOWLEDGE M716-
      M717 : Bool;   // M717-
      Ack_M717 : Bool;   // ACKNOWLEDGE M717-
      M718 : Bool;   // M718-
      Ack_M718 : Bool;   // ACKNOWLEDGE M718-
      M719 : Bool;   // M719-
      Ack_M719 : Bool;   // ACKNOWLEDGE M719-
      M720 : Bool;   // M720-FIXTURE 2 AXIAL LOCATOR LOCATE (READ-IN DISABLE)
      Ack_M720 : Bool;   // ACKNOWLEDGE M720-FIXTURE 2 AXIAL LOCATOR LOCATE (READ-IN DISABLE)
      M721 : Bool;   // M721-FIXTURE 2 AXIAL LOCATOR LOCATE
      Ack_M721 : Bool;   // ACKNOWLEDGE M721-FIXTURE 2 AXIAL LOCATOR LOCATE
      M722 : Bool;   // M722-FIXTURE 2 AXIAL LOCATOR RETURN (READ-IN DISABLE)
      Ack_M722 : Bool;   // ACKNOWLEDGE M722-FIXTURE 2 AXIAL LOCATOR RETURN (READ-IN DISABLE)
      M723 : Bool;   // M723-FIXTURE 2 AXIAL LOCATOR RETURN
      Ack_M723 : Bool;   // ACKNOWLEDGE M723-FIXTURE 2 AXIAL LOCATOR RETURN
      M724 : Bool;   // M724-FIXTURE 2 AXIAL LOCATOR RELEASE PRESSURE (READ-IN DISABLE)
      Ack_M724 : Bool;   // ACKNOWLEDGE M724-FIXTURE 2 AXIAL LOCATOR RELEASE PRESSURE (READ-IN DISABLE)
      M725 : Bool;   // M725-FIXTURE 2 AXIAL LOCATOR LOW PRESSURE (READ-IN DISABLE)
      Ack_M725 : Bool;   // ACKNOWLEDGE M725-FIXTURE 2 AXIAL LOCATOR LOW PRESSURE (READ-IN DISABLE)
      M726 : Bool;   // M726-FIXTURE 2 AXIAL LOCATOR CARRIER ADVANCE (READ-IN DISABLE)
      Ack_M726 : Bool;   // ACKNOWLEDGE M726-FIXTURE 2 AXIAL LOCATOR CARRIER ADVANCE (READ-IN DISABLE)
      M727 : Bool;   // M727-FIXTURE 2 AXIAL LOCATOR CARRIER ADVANCE
      Ack_M727 : Bool;   // ACKNOWLEDGE M727-FIXTURE 2 AXIAL LOCATOR CARRIER ADVANCE
      M728 : Bool;   // M728-FIXTURE 2 AXIAL LOCATOR CARRIER RETURN (READ-IN DISABLE)
      Ack_M728 : Bool;   // ACKNOWLEDGE M728-FIXTURE 2 AXIAL LOCATOR CARRIER RETURN (READ-IN DISABLE)
      M729 : Bool;   // M729-FIXTURE 2 AXIAL LOCATOR CARRIER RETURN
      Ack_M729 : Bool;   // ACKNOWLEDGE M729-FIXTURE 2 AXIAL LOCATOR CARRIER RETURN
      M730 : Bool;   // M730-FIXTURE 2 AXIAL LOCATOR CARRIER RELEASE PRESSURE (READ-IN DISABLE)
      Ack_M730 : Bool;   // ACKNOWLEDGE M730-FIXTURE 2 AXIAL LOCATOR CARRIER RELEASE PRESSURE (READ-IN DISABLE)
      M731 : Bool;   // M731-FIXTURE 2 AXIAL LOCATOR CARRIER LOW PRESSURE (READ-IN DISABLE)
      Ack_M731 : Bool;   // ACKNOWLEDGE M731-FIXTURE 2 AXIAL LOCATOR CARRIER LOW PRESSURE (READ-IN DISABLE)
      M732 : Bool;   // M732-
      Ack_M732 : Bool;   // ACKNOWLEDGE M732-
      M733 : Bool;   // M733-
      Ack_M733 : Bool;   // ACKNOWLEDGE M733-
      M734 : Bool;   // M734-
      Ack_M734 : Bool;   // ACKNOWLEDGE M734-
      M735 : Bool;   // M735-
      Ack_M735 : Bool;   // ACKNOWLEDGE M735-
      M736 : Bool;   // M736-
      Ack_M736 : Bool;   // ACKNOWLEDGE M736-
      M737 : Bool;   // M737-
      Ack_M737 : Bool;   // ACKNOWLEDGE M737-
      M738 : Bool;   // M738-
      Ack_M738 : Bool;   // ACKNOWLEDGE M738-
      M739 : Bool;   // M739-
      Ack_M739 : Bool;   // ACKNOWLEDGE M739-
      M740 : Bool;   // M740-
      Ack_M740 : Bool;   // ACKNOWLEDGE M740-
      M741 : Bool;   // M741-
      Ack_M741 : Bool;   // ACKNOWLEDGE M741-
      M742 : Bool;   // M742-
      Ack_M742 : Bool;   // ACKNOWLEDGE M742-
      M743 : Bool;   // M743-
      Ack_M743 : Bool;   // ACKNOWLEDGE M743-
      M744 : Bool;   // M744-FIXTURE 2 RADIAL LOCATOR LOCATE (READ-IN DISABLE)
      Ack_M744 : Bool;   // ACKNOWLEDGE M744-FIXTURE 2 RADIAL LOCATOR LOCATE (READ-IN DISABLE)
      M745 : Bool;   // M745-FIXTURE 2 RADIAL LOCATOR LOCATE
      Ack_M745 : Bool;   // ACKNOWLEDGE M745-FIXTURE 2 RADIAL LOCATOR LOCATE
      M746 : Bool;   // M746-FIXTURE 2 RADIAL LOCATOR RETURN (READ-IN DISABLE)
      Ack_M746 : Bool;   // ACKNOWLEDGE M746-FIXTURE 2 RADIAL LOCATOR RETURN (READ-IN DISABLE)
      M747 : Bool;   // M747-FIXTURE 2 RADIAL LOCATOR RETURN
      Ack_M747 : Bool;   // ACKNOWLEDGE M747-FIXTURE 2 RADIAL LOCATOR RETURN
      M748 : Bool;   // M748-FIXTURE 2 RADIAL LOCATOR RELEASE PRESSURE (READ-IN DISABLE)
      Ack_M748 : Bool;   // ACKNOWLEDGE M748-FIXTURE 2 RADIAL LOCATOR RELEASE PRESSURE (READ-IN DISABLE)
      M749 : Bool;   // M749-FIXTURE 2 RADIAL LOCATOR LOW PRESSURE (READ-IN DISABLE)
      Ack_M749 : Bool;   // ACKNOWLEDGE M749-FIXTURE 2 RADIAL LOCATOR LOW PRESSURE (READ-IN DISABLE)
      M750 : Bool;   // M750-FIXTURE 2 RADIAL LOCATOR CARRIER ADVANCE (READ-IN DISABLE)
      Ack_M750 : Bool;   // ACKNOWLEDGE M750-FIXTURE 2 RADIAL LOCATOR CARRIER ADVANCE (READ-IN DISABLE)
      M751 : Bool;   // M751-FIXTURE 2 RADIAL LOCATOR CARRIER ADVANCE
      Ack_M751 : Bool;   // ACKNOWLEDGE M751-FIXTURE 2 RADIAL LOCATOR CARRIER ADVANCE
      M752 : Bool;   // M752-FIXTURE 2 RADIAL LOCATOR CARRIER RETURN (READ-IN DISABLE)
      Ack_M752 : Bool;   // ACKNOWLEDGE M752-FIXTURE 2 RADIAL LOCATOR CARRIER RETURN (READ-IN DISABLE)
      M753 : Bool;   // M753-FIXTURE 2 RADIAL LOCATOR CARRIER RETURN
      Ack_M753 : Bool;   // ACKNOWLEDGE M753-FIXTURE 2 RADIAL LOCATOR CARRIER RETURN
      M754 : Bool;   // M754-FIXTURE 2 RADIAL LOCATOR CARRIER RELEASE PRESSURE (READ-IN DISABLE)
      Ack_M754 : Bool;   // ACKNOWLEDGE M754-FIXTURE 2 RADIAL LOCATOR CARRIER RELEASE PRESSURE (READ-IN DISABLE)
      M755 : Bool;   // M755-FIXTURE 2 RADIAL LOCATOR CARRIER LOW PRESSURE (READ-IN DISABLE)
      Ack_M755 : Bool;   // ACKNOWLEDGE M755-FIXTURE 2 RADIAL LOCATOR CARRIER LOW PRESSURE (READ-IN DISABLE)
      M756 : Bool;   // M756-
      Ack_M756 : Bool;   // ACKNOWLEDGE M756-
      M757 : Bool;   // M757-
      Ack_M757 : Bool;   // ACKNOWLEDGE M757-
      M758 : Bool;   // M758-
      Ack_M758 : Bool;   // ACKNOWLEDGE M758-
      M759 : Bool;   // M759-
      Ack_M759 : Bool;   // ACKNOWLEDGE M759-
      M760 : Bool;   // M760-
      Ack_M760 : Bool;   // ACKNOWLEDGE M760-
      M761 : Bool;   // M761-
      Ack_M761 : Bool;   // ACKNOWLEDGE M761-
      M762 : Bool;   // M762-
      Ack_M762 : Bool;   // ACKNOWLEDGE M762-
      M763 : Bool;   // M763-
      Ack_M763 : Bool;   // ACKNOWLEDGE M763-
      M764 : Bool;   // M764-
      Ack_M764 : Bool;   // ACKNOWLEDGE M764-
      M765 : Bool;   // M765-
      Ack_M765 : Bool;   // ACKNOWLEDGE M765-
      M766 : Bool;   // M766-
      Ack_M766 : Bool;   // ACKNOWLEDGE M766-
      M767 : Bool;   // M767-
      Ack_M767 : Bool;   // ACKNOWLEDGE M767-
      M768 : Bool;   // M768-FIXTURE 2 CLAMPING FLANGE CLAMP (READ-IN DISABLE)
      Ack_M768 : Bool;   // ACKNOWLEDGE M768-FIXTURE 2 CLAMPING FLANGE CLAMP (READ-IN DISABLE)
      M769 : Bool;   // M769-FIXTURE 2 CLAMPING FLANGE CLAMP
      Ack_M769 : Bool;   // ACKNOWLEDGE M769-FIXTURE 2 CLAMPING FLANGE CLAMP
      M770 : Bool;   // M770-FIXTURE 2 CLAMPING FLANGE UNCLAMP (READ-IN DISABLE)
      Ack_M770 : Bool;   // ACKNOWLEDGE M770-FIXTURE 2 CLAMPING FLANGE UNCLAMP (READ-IN DISABLE)
      M771 : Bool;   // M771-FIXTURE 2 CLAMPING FLANGE UNCLAMP
      Ack_M771 : Bool;   // ACKNOWLEDGE M771-FIXTURE 2 CLAMPING FLANGE UNCLAMP
      M772 : Bool;   // M772-FIXTURE 2 CLAMPING FLANGE RELEASE PRESSURE (READ-IN DISABLE)
      Ack_M772 : Bool;   // ACKNOWLEDGE M772-FIXTURE 2 CLAMPING FLANGE RELEASE PRESSURE (READ-IN DISABLE)
      M773 : Bool;   // M773-FIXTURE 2 CLAMPING FLANGE LOW PRESSURE (READ-IN DISABLE)
      Ack_M773 : Bool;   // ACKNOWLEDGE M773-FIXTURE 2 CLAMPING FLANGE LOW PRESSURE (READ-IN DISABLE)
      M774 : Bool;   // M774-
      Ack_M774 : Bool;   // ACKNOWLEDGE M774-
      M775 : Bool;   // M775-
      Ack_M775 : Bool;   // ACKNOWLEDGE M775-
      M776 : Bool;   // M776-
      Ack_M776 : Bool;   // ACKNOWLEDGE M776-
      M777 : Bool;   // M777-
      Ack_M777 : Bool;   // ACKNOWLEDGE M777-
      M778 : Bool;   // M778-
      Ack_M778 : Bool;   // ACKNOWLEDGE M778-
      M779 : Bool;   // M779-
      Ack_M779 : Bool;   // ACKNOWLEDGE M779-
      M780 : Bool;   // M780-
      Ack_M780 : Bool;   // ACKNOWLEDGE M780-
      M781 : Bool;   // M781-
      Ack_M781 : Bool;   // ACKNOWLEDGE M781-
      M782 : Bool;   // M782-
      Ack_M782 : Bool;   // ACKNOWLEDGE M782-
      M783 : Bool;   // M783-
      Ack_M783 : Bool;   // ACKNOWLEDGE M783-
      M784 : Bool;   // M784-
      Ack_M784 : Bool;   // ACKNOWLEDGE M784-
      M785 : Bool;   // M785-
      Ack_M785 : Bool;   // ACKNOWLEDGE M785-
      M786 : Bool;   // M786-FIXTURE 2 TAILSTOCK ADVANCE (READ-IN DISABLE)
      Ack_M786 : Bool;   // ACKNOWLEDGE M786-FIXTURE 2 TAILSTOCK ADVANCE (READ-IN DISABLE)
      M787 : Bool;   // M787-FIXTURE 2 TAILSTOCK ADVANCE
      Ack_M787 : Bool;   // ACKNOWLEDGE M787-FIXTURE 2 TAILSTOCK ADVANCE
      M788 : Bool;   // M788-FIXTURE 2 TAILSTOCK RETURN (READ-IN DISABLE)
      Ack_M788 : Bool;   // ACKNOWLEDGE M788-FIXTURE 2 TAILSTOCK RETURN (READ-IN DISABLE)
      M789 : Bool;   // M789-FIXTURE 2 TAILSTOCK RETURN
      Ack_M789 : Bool;   // ACKNOWLEDGE M789-FIXTURE 2 TAILSTOCK RETURN
      M790 : Bool;   // M790-FIXTURE 2 TAILSTOCK RELEASE PRESSURE (READ-IN DISABLE)
      Ack_M790 : Bool;   // ACKNOWLEDGE M790-FIXTURE 2 TAILSTOCK RELEASE PRESSURE (READ-IN DISABLE)
      M791 : Bool;   // M791-FIXTURE 2 TAILSTOCK LOW PRESSURE (READ-IN DISABLE)
      Ack_M791 : Bool;   // ACKNOWLEDGE M791-FIXTURE 2 TAILSTOCK LOW PRESSURE (READ-IN DISABLE)
      M792 : Bool;   // M792-
      Ack_M792 : Bool;   // ACKNOWLEDGE M792-
      M793 : Bool;   // M793-
      Ack_M793 : Bool;   // ACKNOWLEDGE M793-
      M794 : Bool;   // M794-
      Ack_M794 : Bool;   // ACKNOWLEDGE M794-
      M795 : Bool;   // M795-
      Ack_M795 : Bool;   // ACKNOWLEDGE M795-
      M796 : Bool;   // M796-
      Ack_M796 : Bool;   // ACKNOWLEDGE M796-
      M797 : Bool;   // M797-
      Ack_M797 : Bool;   // ACKNOWLEDGE M797-
      M798 : Bool;   // M798-FIXTURE 2 SHIFTING DEVICE LOCATE (READ-IN DISABLE)
      Ack_M798 : Bool;   // ACKNOWLEDGE M798-FIXTURE 2 SHIFTING DEVICE LOCATE (READ-IN DISABLE)
      M799 : Bool;   // M799-FIXTURE 2 SHIFTING DEVICE LOCATE
      Ack_M799 : Bool;   // ACKNOWLEDGE M799-FIXTURE 2 SHIFTING DEVICE LOCATE
      M800 : Bool;   // M800-FIXTURE 2 SHIFTING DEVICE RETURN (READ-IN DISABLE)
      Ack_M800 : Bool;   // ACKNOWLEDGE M800-FIXTURE 2 SHIFTING DEVICE RETURN (READ-IN DISABLE)
      M801 : Bool;   // M801-FIXTURE 2 SHIFTING DEVICE RETURN
      Ack_M801 : Bool;   // ACKNOWLEDGE M801-FIXTURE 2 SHIFTING DEVICE RETURN
      M802 : Bool;   // M802-FIXTURE 2 SHIFTING DEVICE RELEASE PRESSURE (READ-IN DISABLE)
      Ack_M802 : Bool;   // ACKNOWLEDGE M802-FIXTURE 2 SHIFTING DEVICE RELEASE PRESSURE (READ-IN DISABLE)
      M803 : Bool;   // M803-FIXTURE 2 SHIFTING DEVICE LOW PRESSURE (READ-IN DISABLE)
      Ack_M803 : Bool;   // ACKNOWLEDGE M803-FIXTURE 2 SHIFTING DEVICE LOW PRESSURE (READ-IN DISABLE)
      M804 : Bool;   // M804-FIXTURE 2 BLOCKING DEVICE BLOCK (READ-IN DISABLE)
      Ack_M804 : Bool;   // ACKNOWLEDGE M804-FIXTURE 2 BLOCKING DEVICE BLOCK (READ-IN DISABLE)
      M805 : Bool;   // M805-FIXTURE 2 BLOCKING DEVICE BLOCK
      Ack_M805 : Bool;   // ACKNOWLEDGE M805-FIXTURE 2 BLOCKING DEVICE BLOCK
      M806 : Bool;   // M806-FIXTURE 2 BLOCKING DEVICE UNBLOCK (READ-IN DISABLE)
      Ack_M806 : Bool;   // ACKNOWLEDGE M806-FIXTURE 2 BLOCKING DEVICE UNBLOCK (READ-IN DISABLE)
      M807 : Bool;   // M807-FIXTURE 2 BLOCKING DEVICE UNBLOCK
      Ack_M807 : Bool;   // ACKNOWLEDGE M807-FIXTURE 2 BLOCKING DEVICE UNBLOCK
      M808 : Bool;   // M808-FIXTURE 2 BLOCKING DEVICE RELEASE PRESSURE (READ-IN DISABLE)
      Ack_M808 : Bool;   // ACKNOWLEDGE M808-FIXTURE 2 BLOCKING DEVICE RELEASE PRESSURE (READ-IN DISABLE)
      M809 : Bool;   // M809-FIXTURE 2 BLOCKING DEVICE LOW PRESSURE (READ-IN DISABLE)
      Ack_M809 : Bool;   // ACKNOWLEDGE M809-FIXTURE 2 BLOCKING DEVICE LOW PRESSURE (READ-IN DISABLE)
      M810 : Bool;   // M810-FIXTURE 2 VIBRATION DAMPER CLAMP (READ-IN DISABLE)
      Ack_M810 : Bool;   // ACKNOWLEDGE M810-FIXTURE 2 VIBRATION DAMPER CLAMP (READ-IN DISABLE)
      M811 : Bool;   // M811-FIXTURE 2 VIBRATION DAMPER CLAMP
      Ack_M811 : Bool;   // ACKNOWLEDGE M811-FIXTURE 2 VIBRATION DAMPER CLAMP
      M812 : Bool;   // M812-FIXTURE 2 VIBRATION DAMPER UNCLAMP (READ-IN DISABLE)
      Ack_M812 : Bool;   // ACKNOWLEDGE M812-FIXTURE 2 VIBRATION DAMPER UNCLAMP (READ-IN DISABLE)
      M813 : Bool;   // M813-FIXTURE 2 VIBRATION DAMPER UNCLAMP
      Ack_M813 : Bool;   // ACKNOWLEDGE M813-FIXTURE 2 VIBRATION DAMPER UNCLAMP
      M814 : Bool;   // M814-FIXTURE 2 VIBRATION DAMPER RELEASE PRESSURE (READ-IN DISABLE)
      Ack_M814 : Bool;   // ACKNOWLEDGE M814-FIXTURE 2 VIBRATION DAMPER RELEASE PRESSURE (READ-IN DISABLE)
      M815 : Bool;   // M815-FIXTURE 2 VIBRATION DAMPER LOW PRESSURE (READ-IN DISABLE)
      Ack_M815 : Bool;   // ACKNOWLEDGE M815-FIXTURE 2 VIBRATION DAMPER LOW PRESSURE (READ-IN DISABLE)
      M816 : Bool;   // M816-
      Ack_M816 : Bool;   // ACKNOWLEDGE M816-
      M817 : Bool;   // M817-
      Ack_M817 : Bool;   // ACKNOWLEDGE M817-
      M818 : Bool;   // M818-
      Ack_M818 : Bool;   // ACKNOWLEDGE M818-
      M819 : Bool;   // M819-
      Ack_M819 : Bool;   // ACKNOWLEDGE M819-
      M820 : Bool;   // M820-
      Ack_M820 : Bool;   // ACKNOWLEDGE M820-
      M821 : Bool;   // M821-
      Ack_M821 : Bool;   // ACKNOWLEDGE M821-
      M822 : Bool;   // M822-
      Ack_M822 : Bool;   // ACKNOWLEDGE M822-
      M823 : Bool;   // M823-
      Ack_M823 : Bool;   // ACKNOWLEDGE M823-
      M824 : Bool;   // M824-
      Ack_M824 : Bool;   // ACKNOWLEDGE M824-
      M825 : Bool;   // M825-
      Ack_M825 : Bool;   // ACKNOWLEDGE M825-
      M826 : Bool;   // M826-
      Ack_M826 : Bool;   // ACKNOWLEDGE M826-
      M827 : Bool;   // M827-
      Ack_M827 : Bool;   // ACKNOWLEDGE M827-
      M828 : Bool;   // M828-FIXTURE 2 JAW CHUCK CLAMP (READ-IN DISABLE)
      Ack_M828 : Bool;   // ACKNOWLEDGE M828-FIXTURE 2 JAW CHUCK CLAMP (READ-IN DISABLE)
      M829 : Bool;   // M829-FIXTURE 2 JAW CHUCK CLAMP
      Ack_M829 : Bool;   // ACKNOWLEDGE M829-FIXTURE 2 JAW CHUCK CLAMP
      M830 : Bool;   // M830-FIXTURE 2 JAW CHUCK UNCLAMP (READ-IN DISABLE)
      Ack_M830 : Bool;   // ACKNOWLEDGE M830-FIXTURE 2 JAW CHUCK UNCLAMP (READ-IN DISABLE)
      M831 : Bool;   // M831-FIXTURE 2 JAW CHUCK UNCLAMP
      Ack_M831 : Bool;   // ACKNOWLEDGE M831-FIXTURE 2 JAW CHUCK UNCLAMP
      M832 : Bool;   // M832-FIXTURE 2 JAW CHUCK RELEASE PRESSURE (READ-IN DISABLE)
      Ack_M832 : Bool;   // ACKNOWLEDGE M832-FIXTURE 2 JAW CHUCK RELEASE PRESSURE (READ-IN DISABLE)
      M833 : Bool;   // M833-FIXTURE 2 JAW CHUCK LOW CLAMP (READ-IN DISABLE)
      Ack_M833 : Bool;   // ACKNOWLEDGE M833-FIXTURE 2 JAW CHUCK LOW CLAMP (READ-IN DISABLE)
      M834 : Bool;   // M834-
      Ack_M834 : Bool;   // ACKNOWLEDGE M834-
      M835 : Bool;   // M835-
      Ack_M835 : Bool;   // ACKNOWLEDGE M835-
      M836 : Bool;   // M836-
      Ack_M836 : Bool;   // ACKNOWLEDGE M836-
      M837 : Bool;   // M837-
      Ack_M837 : Bool;   // ACKNOWLEDGE M837-
      M838 : Bool;   // M838-
      Ack_M838 : Bool;   // ACKNOWLEDGE M838-
      M839 : Bool;   // M839-
      Ack_M839 : Bool;   // ACKNOWLEDGE M839-
      M840 : Bool;   // M840-
      Ack_M840 : Bool;   // ACKNOWLEDGE M840-
      M841 : Bool;   // M841-
      Ack_M841 : Bool;   // ACKNOWLEDGE M841-
      M842 : Bool;   // M842-
      Ack_M842 : Bool;   // ACKNOWLEDGE M842-
      M843 : Bool;   // M843-
      Ack_M843 : Bool;   // ACKNOWLEDGE M843-
      M844 : Bool;   // M844-
      Ack_M844 : Bool;   // ACKNOWLEDGE M844-
      M845 : Bool;   // M845-
      Ack_M845 : Bool;   // ACKNOWLEDGE M845-
      M846 : Bool;   // M846-FIXTURE 2 CENTRAL JAW CHUCK CLAMP (READ-IN DISABLE)
      Ack_M846 : Bool;   // ACKNOWLEDGE M846-FIXTURE 2 CENTRAL JAW CHUCK CLAMP (READ-IN DISABLE)
      M847 : Bool;   // M847-FIXTURE 2 CENTRAL JAW CHUCK CLAMP
      Ack_M847 : Bool;   // ACKNOWLEDGE M847-FIXTURE 2 CENTRAL JAW CHUCK CLAMP
      M848 : Bool;   // M848-FIXTURE 2 CENTRAL JAW CHUCK UNCLAMP (READ-IN DISABLE)
      Ack_M848 : Bool;   // ACKNOWLEDGE M848-FIXTURE 2 CENTRAL JAW CHUCK UNCLAMP (READ-IN DISABLE)
      M849 : Bool;   // M849-FIXTURE 2 CENTRAL JAW CHUCK UNCLAMP
      Ack_M849 : Bool;   // ACKNOWLEDGE M849-FIXTURE 2 CENTRAL JAW CHUCK UNCLAMP
      M850 : Bool;   // M850-FIXTURE 2 CENTRAL JAW CHUCK RELEASE PRESSURE (READ-IN DISABLE)
      Ack_M850 : Bool;   // ACKNOWLEDGE M850-FIXTURE 2 CENTRAL JAW CHUCK RELEASE PRESSURE (READ-IN DISABLE)
      M851 : Bool;   // M851-FIXTURE 2 CENTRAL JAW CHUCK LOW CLAMP (READ-IN DISABLE)
      Ack_M851 : Bool;   // ACKNOWLEDGE M851-FIXTURE 2 CENTRAL JAW CHUCK LOW CLAMP (READ-IN DISABLE)
      M852 : Bool;   // M852-
      Ack_M852 : Bool;   // ACKNOWLEDGE M852-
      M853 : Bool;   // M853-
      Ack_M853 : Bool;   // ACKNOWLEDGE M853-
      M854 : Bool;   // M854-
      Ack_M854 : Bool;   // ACKNOWLEDGE M854-
      M855 : Bool;   // M855-
      Ack_M855 : Bool;   // ACKNOWLEDGE M855-
      M856 : Bool;   // M856-
      Ack_M856 : Bool;   // ACKNOWLEDGE M856-
      M857 : Bool;   // M857-
      Ack_M857 : Bool;   // ACKNOWLEDGE M857-
      M858 : Bool;   // M858-
      Ack_M858 : Bool;   // ACKNOWLEDGE M858-
      M859 : Bool;   // M859-
      Ack_M859 : Bool;   // ACKNOWLEDGE M859-
      M860 : Bool;   // M860-
      Ack_M860 : Bool;   // ACKNOWLEDGE M860-
      M861 : Bool;   // M861-
      Ack_M861 : Bool;   // ACKNOWLEDGE M861-
      M862 : Bool;   // M862-
      Ack_M862 : Bool;   // ACKNOWLEDGE M862-
      M863 : Bool;   // M863-
      Ack_M863 : Bool;   // ACKNOWLEDGE M863-
      M864 : Bool;   // M864-FIXTURE 2 JAW CHUCK B CLAMP (READ-IN DISABLE)
      Ack_M864 : Bool;   // ACKNOWLEDGE M864-FIXTURE 2 JAW CHUCK B CLAMP (READ-IN DISABLE)
      M865 : Bool;   // M865-FIXTURE 2 JAW CHUCK B CLAMP
      Ack_M865 : Bool;   // ACKNOWLEDGE M865-FIXTURE 2 JAW CHUCK B CLAMP
      M866 : Bool;   // M866-FIXTURE 2 JAW CHUCK B UNCLAMP (READ-IN DISABLE)
      Ack_M866 : Bool;   // ACKNOWLEDGE M866-FIXTURE 2 JAW CHUCK B UNCLAMP (READ-IN DISABLE)
      M867 : Bool;   // M867-FIXTURE 2 JAW CHUCK B UNCLAMP
      Ack_M867 : Bool;   // ACKNOWLEDGE M867-FIXTURE 2 JAW CHUCK B UNCLAMP
      M868 : Bool;   // M868-FIXTURE 2 JAW CHUCK B RELEASE PRESSURE
      Ack_M868 : Bool;   // ACKNOWLEDGE M868-FIXTURE 2 JAW CHUCK B RELEASE PRESSURE
      M869 : Bool;   // M869-FIXTURE 2 JAW CHUCK B LOW PRESSURE
      Ack_M869 : Bool;   // ACKNOWLEDGE M869-FIXTURE 2 JAW CHUCK B LOW PRESSURE
      M870 : Bool;   // M870-FIXTURE 2 ROTARY JAW CHUCK CLAMP (READ-IN DISABLE)
      Ack_M870 : Bool;   // ACKNOWLEDGE M870-FIXTURE 2 ROTARY JAW CHUCK CLAMP (READ-IN DISABLE)
      M871 : Bool;   // M871-FIXTURE 2 ROTARY JAW CHUCK CLAMP
      Ack_M871 : Bool;   // ACKNOWLEDGE M871-FIXTURE 2 ROTARY JAW CHUCK CLAMP
      M872 : Bool;   // M872-FIXTURE 2 ROTARY JAW CHUCK UNCLAMP (READ-IN DISABLE)
      Ack_M872 : Bool;   // ACKNOWLEDGE M872-FIXTURE 2 ROTARY JAW CHUCK UNCLAMP (READ-IN DISABLE)
      M873 : Bool;   // M873-FIXTURE 2 ROTARY JAW CHUCK UNCLAMP
      Ack_M873 : Bool;   // ACKNOWLEDGE M873-FIXTURE 2 ROTARY JAW CHUCK UNCLAMP
      M874 : Bool;   // M874-FIXTURE 2 ROTARY JAW CHUCK RELEASE PRESSURE (READ-IN DISABLE)
      Ack_M874 : Bool;   // ACKNOWLEDGE M874-FIXTURE 2 ROTARY JAW CHUCK RELEASE PRESSURE (READ-IN DISABLE)
      M875 : Bool;   // M875-FIXTURE 2 ROTARY JAW CHUCK LOW PRESSURE (READ-IN DISABLE)
      Ack_M875 : Bool;   // ACKNOWLEDGE M875-FIXTURE 2 ROTARY JAW CHUCK LOW PRESSURE (READ-IN DISABLE)
      M876 : Bool;   // M876-
      Ack_M876 : Bool;   // ACKNOWLEDGE M876-
      M877 : Bool;   // M877-
      Ack_M877 : Bool;   // ACKNOWLEDGE M877-
      M878 : Bool;   // M878-
      Ack_M878 : Bool;   // ACKNOWLEDGE M878-
      M879 : Bool;   // M879-
      Ack_M879 : Bool;   // ACKNOWLEDGE M879-
      M880 : Bool;   // M880-
      Ack_M880 : Bool;   // ACKNOWLEDGE M880-
      M881 : Bool;   // M881-
      Ack_M881 : Bool;   // ACKNOWLEDGE M881-
      M882 : Bool;   // M882-
      Ack_M882 : Bool;   // ACKNOWLEDGE M882-
      M883 : Bool;   // M883-
      Ack_M883 : Bool;   // ACKNOWLEDGE M883-
      M884 : Bool;   // M884-
      Ack_M884 : Bool;   // ACKNOWLEDGE M884-
      M885 : Bool;   // M885-
      Ack_M885 : Bool;   // ACKNOWLEDGE M885-
      M886 : Bool;   // M886-
      Ack_M886 : Bool;   // ACKNOWLEDGE M886-
      M887 : Bool;   // M887-
      Ack_M887 : Bool;   // ACKNOWLEDGE M887-
      M888 : Bool;   // M888-FIXTURE 2 REMOVABLE STOP ADVANCE (READ-IN DISABLE)
      Ack_M888 : Bool;   // ACKNOWLEDGE M888-FIXTURE 2 REMOVABLE STOP ADVANCE (READ-IN DISABLE)
      M889 : Bool;   // M889-FIXTURE 2 REMOVABLE STOP ADVANCE
      Ack_M889 : Bool;   // ACKNOWLEDGE M889-FIXTURE 2 REMOVABLE STOP ADVANCE
      M890 : Bool;   // M890-FIXTURE 2 REMOVABLE STOP RETURN (READ-IN DISABLE)
      Ack_M890 : Bool;   // ACKNOWLEDGE M890-FIXTURE 2 REMOVABLE STOP RETURN (READ-IN DISABLE)
      M891 : Bool;   // M891-FIXTURE 2 REMOVABLE STOP RETURN
      Ack_M891 : Bool;   // ACKNOWLEDGE M891-FIXTURE 2 REMOVABLE STOP RETURN
      M892 : Bool;   // M892-FIXTURE 2 REMOVABLE STOP RELEASE PRESSURE (READ-IN DISABLE)
      Ack_M892 : Bool;   // ACKNOWLEDGE M892-FIXTURE 2 REMOVABLE STOP RELEASE PRESSURE (READ-IN DISABLE)
      M893 : Bool;   // M893-FIXTURE 2 REMOVABLE STOP LOW PRESSURE (READ-IN DISABLE)
      Ack_M893 : Bool;   // ACKNOWLEDGE M893-FIXTURE 2 REMOVABLE STOP LOW PRESSURE (READ-IN DISABLE)
      M894 : Bool;   // M894-
      Ack_M894 : Bool;   // ACKNOWLEDGE M894-
      M895 : Bool;   // M895-
      Ack_M895 : Bool;   // ACKNOWLEDGE M895-
      M896 : Bool;   // M896-
      Ack_M896 : Bool;   // ACKNOWLEDGE M896-
      M897 : Bool;   // M897-
      Ack_M897 : Bool;   // ACKNOWLEDGE M897-
      M898 : Bool;   // M898-
      Ack_M898 : Bool;   // ACKNOWLEDGE M898-
      M899 : Bool;   // M899-
      Ack_M899 : Bool;   // ACKNOWLEDGE M899-
      M900 : Bool;   // M900-
      Ack_M900 : Bool;   // ACKNOWLEDGE M900-
      M901 : Bool;   // M901-
      Ack_M901 : Bool;   // ACKNOWLEDGE M901-
      M902 : Bool;   // M902-
      Ack_M902 : Bool;   // ACKNOWLEDGE M902-
      M903 : Bool;   // M903-
      Ack_M903 : Bool;   // ACKNOWLEDGE M903-
      M904 : Bool;   // M904-
      Ack_M904 : Bool;   // ACKNOWLEDGE M904-
      M905 : Bool;   // M905-
      Ack_M905 : Bool;   // ACKNOWLEDGE M905-
      M906 : Bool;   // M906-
      Ack_M906 : Bool;   // ACKNOWLEDGE M906-
      M907 : Bool;   // M907-
      Ack_M907 : Bool;   // ACKNOWLEDGE M907-
      M908 : Bool;   // M908-
      Ack_M908 : Bool;   // ACKNOWLEDGE M908-
      M909 : Bool;   // M909-
      Ack_M909 : Bool;   // ACKNOWLEDGE M909-
      M910 : Bool;   // M910-
      Ack_M910 : Bool;   // ACKNOWLEDGE M910-
      M911 : Bool;   // M911-
      Ack_M911 : Bool;   // ACKNOWLEDGE M911-
      M912 : Bool;   // M912-
      Ack_M912 : Bool;   // ACKNOWLEDGE M912-
      M913 : Bool;   // M913-
      Ack_M913 : Bool;   // ACKNOWLEDGE M913-
      M914 : Bool;   // M914-
      Ack_M914 : Bool;   // ACKNOWLEDGE M914-
      M915 : Bool;   // M915-
      Ack_M915 : Bool;   // ACKNOWLEDGE M915-
      M916 : Bool;   // M916-
      Ack_M916 : Bool;   // ACKNOWLEDGE M916-
      M917 : Bool;   // M917-
      Ack_M917 : Bool;   // ACKNOWLEDGE M917-
      M918 : Bool;   // M918-
      Ack_M918 : Bool;   // ACKNOWLEDGE M918-
      M919 : Bool;   // M919-
      Ack_M919 : Bool;   // ACKNOWLEDGE M919-
      M920 : Bool;   // M920-
      Ack_M920 : Bool;   // ACKNOWLEDGE M920-
      M921 : Bool;   // M921-
      Ack_M921 : Bool;   // ACKNOWLEDGE M921-
      M922 : Bool;   // M922-
      Ack_M922 : Bool;   // ACKNOWLEDGE M922-
      M923 : Bool;   // M923-
      Ack_M923 : Bool;   // ACKNOWLEDGE M923-
      M924 : Bool;   // M924-
      Ack_M924 : Bool;   // ACKNOWLEDGE M924-
      M925 : Bool;   // M925-
      Ack_M925 : Bool;   // ACKNOWLEDGE M925-
      M926 : Bool;   // M926-
      Ack_M926 : Bool;   // ACKNOWLEDGE M926-
      M927 : Bool;   // M927-
      Ack_M927 : Bool;   // ACKNOWLEDGE M927-
      M928 : Bool;   // M928-
      Ack_M928 : Bool;   // ACKNOWLEDGE M928-
      M929 : Bool;   // M929-
      Ack_M929 : Bool;   // ACKNOWLEDGE M929-
      M930 : Bool;   // M930-
      Ack_M930 : Bool;   // ACKNOWLEDGE M930-
      M931 : Bool;   // M931-
      Ack_M931 : Bool;   // ACKNOWLEDGE M931-
      M932 : Bool;   // M932-
      Ack_M932 : Bool;   // ACKNOWLEDGE M932-
      M933 : Bool;   // M933-
      Ack_M933 : Bool;   // ACKNOWLEDGE M933-
      M934 : Bool;   // M934-
      Ack_M934 : Bool;   // ACKNOWLEDGE M934-
      M935 : Bool;   // M935-
      Ack_M935 : Bool;   // ACKNOWLEDGE M935-
      M936 : Bool;   // M936-
      Ack_M936 : Bool;   // ACKNOWLEDGE M936-
      M937 : Bool;   // M937-
      Ack_M937 : Bool;   // ACKNOWLEDGE M937-
      M938 : Bool;   // M938-
      Ack_M938 : Bool;   // ACKNOWLEDGE M938-
      M939 : Bool;   // M939-
      Ack_M939 : Bool;   // ACKNOWLEDGE M939-
      M940 : Bool;   // M940-
      Ack_M940 : Bool;   // ACKNOWLEDGE M940-
      M941 : Bool;   // M941-
      Ack_M941 : Bool;   // ACKNOWLEDGE M941-
      M942 : Bool;   // M942-
      Ack_M942 : Bool;   // ACKNOWLEDGE M942-
      M943 : Bool;   // M943-
      Ack_M943 : Bool;   // ACKNOWLEDGE M943-
      M944 : Bool;   // M944-
      Ack_M944 : Bool;   // ACKNOWLEDGE M944-
      M945 : Bool;   // M945-
      Ack_M945 : Bool;   // ACKNOWLEDGE M945-
      M946 : Bool;   // M946-
      Ack_M946 : Bool;   // ACKNOWLEDGE M946-
      M947 : Bool;   // M947-
      Ack_M947 : Bool;   // ACKNOWLEDGE M947-
      M948 : Bool;   // M948-
      Ack_M948 : Bool;   // ACKNOWLEDGE M948-
      M949 : Bool;   // M949-
      Ack_M949 : Bool;   // ACKNOWLEDGE M949-
      M950 : Bool;   // M950-
      Ack_M950 : Bool;   // ACKNOWLEDGE M950-
      M951 : Bool;   // M951-
      Ack_M951 : Bool;   // ACKNOWLEDGE M951-
      M952 : Bool;   // M952-
      Ack_M952 : Bool;   // ACKNOWLEDGE M952-
      M953 : Bool;   // M953-
      Ack_M953 : Bool;   // ACKNOWLEDGE M953-
      M954 : Bool;   // M954-
      Ack_M954 : Bool;   // ACKNOWLEDGE M954-
      M955 : Bool;   // M955-
      Ack_M955 : Bool;   // ACKNOWLEDGE M955-
      M956 : Bool;   // M956-
      Ack_M956 : Bool;   // ACKNOWLEDGE M956-
      M957 : Bool;   // M957-
      Ack_M957 : Bool;   // ACKNOWLEDGE M957-
      M958 : Bool;   // M958-
      Ack_M958 : Bool;   // ACKNOWLEDGE M958-
      M959 : Bool;   // M959-
      Ack_M959 : Bool;   // ACKNOWLEDGE M959-
      M960 : Bool;   // M960-
      Ack_M960 : Bool;   // ACKNOWLEDGE M960-
      M961 : Bool;   // M961-
      Ack_M961 : Bool;   // ACKNOWLEDGE M961-
      M962 : Bool;   // M962-
      Ack_M962 : Bool;   // ACKNOWLEDGE M962-
      M963 : Bool;   // M963-
      Ack_M963 : Bool;   // ACKNOWLEDGE M963-
      M964 : Bool;   // M964-
      Ack_M964 : Bool;   // ACKNOWLEDGE M964-
      M965 : Bool;   // M965-
      Ack_M965 : Bool;   // ACKNOWLEDGE M965-
      M966 : Bool;   // M966-
      Ack_M966 : Bool;   // ACKNOWLEDGE M966-
      M967 : Bool;   // M967-
      Ack_M967 : Bool;   // ACKNOWLEDGE M967-
      M968 : Bool;   // M968-
      Ack_M968 : Bool;   // ACKNOWLEDGE M968-
      M969 : Bool;   // M969-
      Ack_M969 : Bool;   // ACKNOWLEDGE M969-
      M970 : Bool;   // M970-
      Ack_M970 : Bool;   // ACKNOWLEDGE M970-
      M971 : Bool;   // M971-
      Ack_M971 : Bool;   // ACKNOWLEDGE M971-
      M972 : Bool;   // M972-
      Ack_M972 : Bool;   // ACKNOWLEDGE M972-
      M973 : Bool;   // M973-
      Ack_M973 : Bool;   // ACKNOWLEDGE M973-
      M974 : Bool;   // M974-
      Ack_M974 : Bool;   // ACKNOWLEDGE M974-
      M975 : Bool;   // M975-
      Ack_M975 : Bool;   // ACKNOWLEDGE M975-
      M976 : Bool;   // M976-
      Ack_M976 : Bool;   // ACKNOWLEDGE M976-
      M977 : Bool;   // M977-
      Ack_M977 : Bool;   // ACKNOWLEDGE M977-
      M978 : Bool;   // M978-
      Ack_M978 : Bool;   // ACKNOWLEDGE M978-
      M979 : Bool;   // M979-
      Ack_M979 : Bool;   // ACKNOWLEDGE M979-
      M980 : Bool;   // M980-
      Ack_M980 : Bool;   // ACKNOWLEDGE M980-
      M981 : Bool;   // M981-
      Ack_M981 : Bool;   // ACKNOWLEDGE M981-
      M982 : Bool;   // M982-
      Ack_M982 : Bool;   // ACKNOWLEDGE M982-
      M983 : Bool;   // M983-
      Ack_M983 : Bool;   // ACKNOWLEDGE M983-
      M984 : Bool;   // M984-
      Ack_M984 : Bool;   // ACKNOWLEDGE M984-
      M985 : Bool;   // M985-
      Ack_M985 : Bool;   // ACKNOWLEDGE M985-
      M986 : Bool;   // M986-
      Ack_M986 : Bool;   // ACKNOWLEDGE M986-
      M987 : Bool;   // M987-
      Ack_M987 : Bool;   // ACKNOWLEDGE M987-
      M988 : Bool;   // M988-
      Ack_M988 : Bool;   // ACKNOWLEDGE M988-
      M989 : Bool;   // M989-
      Ack_M989 : Bool;   // ACKNOWLEDGE M989-
      M990 : Bool;   // M990-
      Ack_M990 : Bool;   // ACKNOWLEDGE M990-
      M991 : Bool;   // M991-
      Ack_M991 : Bool;   // ACKNOWLEDGE M991-
      M992 : Bool;   // M992-
      Ack_M992 : Bool;   // ACKNOWLEDGE M992-
      M993 : Bool;   // M993-
      Ack_M993 : Bool;   // ACKNOWLEDGE M993-
      M994 : Bool;   // M994-
      Ack_M994 : Bool;   // ACKNOWLEDGE M994-
      M995 : Bool;   // M995-
      Ack_M995 : Bool;   // ACKNOWLEDGE M995-
      M996 : Bool;   // M996-
      Ack_M996 : Bool;   // ACKNOWLEDGE M996-
      M997 : Bool;   // M997-
      Ack_M997 : Bool;   // ACKNOWLEDGE M997-
      M998 : Bool;   // M998-
      Ack_M998 : Bool;   // ACKNOWLEDGE M998-
      M999 : Bool;   // M999-
      Ack_M999 : Bool;   // ACKNOWLEDGE M999-
   END_STRUCT;
END_TYPE
